# B&R Automation Studio project FASTorySystems (part 3)

### IoMap.iom - 5APC4100_TGL2_000/IoMap.iom
```iecst
VAR_CONFIG
	Cyclic#1.::gCommInput.Array[0] AT %IW."8FLM01.0000.00I-1".EPL_FB_IN_0_I2007_S01;
	Cyclic#1.::gCommInput.Array[1] AT %IW."8FLM01.0000.00I-1".EPL_FB_IN_1_I2007_S02;
	Cyclic#1.::gCommInput.Array[2] AT %IW."8FLM01.0000.00I-1".EPL_FB_IN_2_I2007_S03;
	Cyclic#1.::gCommInput.Array[3] AT %IW."8FLM01.0000.00I-1".EPL_FB_IN_3_I2007_S04;
	Cyclic#1.::gCommInput.Array[4] AT %IW."8FLM01.0000.00I-1".EPL_FB_IN_4_I2007_S05;
	Cyclic#1.::gCommInput.Array[5] AT %IW."8FLM01.0000.00I-1".EPL_FB_IN_5_I2007_S06;
	Cyclic#1.::gCommInput.Array[6] AT %IW."8FLM01.0000.00I-1".EPL_FB_IN_6_I2007_S07;
	Cyclic#1.::gCommInput.Array[7] AT %IW."8FLM01.0000.00I-1".EPL_FB_IN_7_I2007_S08;
	Cyclic#1.::gCommInput.Array[8] AT %IW."8FLM01.0000.00I-1".EPL_FB_IN_8_I2007_S09;
	Cyclic#1.::gCommInput.Array[9] AT %IW."8FLM01.0000.00I-1".EPL_FB_IN_9_I2007_S0A;
	Cyclic#1.::gCommInput.Array[10] AT %IW."8FLM01.0000.00I-1".EPL_FB_IN_10_I2007_S0B;
	Cyclic#1.::gCommInput.Array[11] AT %IW."8FLM01.0000.00I-1".EPL_FB_IN_11_I2007_S0C;
	Cyclic#1.::gCommInput.Array[12] AT %IW."8FLM01.0000.00I-1".EPL_FB_IN_12_I2007_S0D;
	Cyclic#1.::gCommInput.Array[13] AT %IW."8FLM01.0000.00I-1".EPL_FB_IN_13_I2007_S0E;
	Cyclic#1.::gCommInput.Array[14] AT %IW."8FLM01.0000.00I-1".EPL_FB_IN_14_I2007_S0F;
	Cyclic#1.::gCommInput.Array[15] AT %IW."8FLM01.0000.00I-1".EPL_FB_IN_15_I2007_S10;
	Cyclic#1.::gCommInput.Array[16] AT %IW."8FLM01.0000.00I-1".EPL_FB_IN_16_I2007_S11;
	Cyclic#1.::gCommInput.Array[17] AT %IW."8FLM01.0000.00I-1".EPL_FB_IN_17_I2007_S12;
	Cyclic#1.::gCommInput.Array[18] AT %IW."8FLM01.0000.00I-1".EPL_FB_IN_18_I2007_S13;
	Cyclic#1.::gCommInput.Array[19] AT %IW."8FLM01.0000.00I-1".EPL_FB_IN_19_I2007_S14;
	Cyclic#1.::gCommInput.Array[20] AT %IW."8FLM01.0000.00I-1".EPL_FB_IN_20_I2007_S15;
	Cyclic#1.::gCommInput.Array[21] AT %IW."8FLM01.0000.00I-1".EPL_FB_IN_21_I2007_S16;
	Cyclic#1.::gCommInput.Array[22] AT %IW."8FLM01.0000.00I-1".EPL_FB_IN_22_I2007_S17;
	Cyclic#1.::gCommInput.Array[23] AT %IW."8FLM01.0000.00I-1".EPL_FB_IN_23_I2007_S18;
	Cyclic#1.::gCommInput.Array[24] AT %IW."8FLM01.0000.00I-1".EPL_FB_IN_24_I2007_S19;
	Cyclic#1.::gCommInput.Array[25] AT %IW."8FLM01.0000.00I-1".EPL_FB_IN_25_I2007_S1A;
	Cyclic#1.::gCommInput.Array[26] AT %IW."8FLM01.0000.00I-1".EPL_FB_IN_26_I2007_S1B;
	Cyclic#1.::gCommInput.Array[27] AT %IW."8FLM01.0000.00I-1".EPL_FB_IN_27_I2007_S1C;
	Cyclic#1.::gCommInput.Array[28] AT %IW."8FLM01.0000.00I-1".EPL_FB_IN_28_I2007_S1D;
	Cyclic#1.::gCommInput.Array[29] AT %IW."8FLM01.0000.00I-1".EPL_FB_IN_29_I2007_S1E;
	Cyclic#1.::gCommInput.Array[30] AT %IW."8FLM01.0000.00I-1".EPL_FB_IN_30_I2007_S1F;
	Cyclic#1.::gCommInput.Array[31] AT %IW."8FLM01.0000.00I-1".EPL_FB_IN_31_I2007_S20;
	Cyclic#1.::gCommInput.Array[32] AT %IW."8FLM01.0000.00I-1".EPL_FB_IN_32_I2007_S21;
	Cyclic#1.::gCommInput.Array[33] AT %IW."8FLM01.0000.00I-1".EPL_FB_IN_33_I2007_S22;
	Cyclic#1.::gCommInput.Array[34] AT %IW."8FLM01.0000.00I-1".EPL_FB_IN_34_I2007_S23;
	Cyclic#1.::gCommInput.Array[35] AT %IW."8FLM01.0000.00I-1".EPL_FB_IN_35_I2007_S24;
	Cyclic#1.::gCommInput.Array[36] AT %IW."8FLM01.0000.00I-1".EPL_FB_IN_36_I2007_S25;
	Cyclic#1.::gCommInput.Array[37] AT %IW."8FLM01.0000.00I-1".EPL_FB_IN_37_I2007_S26;
	Cyclic#1.::gCommInput.Array[38] AT %IW."8FLM01.0000.00I-1".EPL_FB_IN_38_I2007_S27;
	Cyclic#1.::gCommInput.Array[39] AT %IW."8FLM01.0000.00I-1".EPL_FB_IN_39_I2007_S28;
	Cyclic#1.::gCommInput.Array[40] AT %IW."8FLM01.0000.00I-1".EPL_FB_IN_40_I2007_S29;
	Cyclic#1.::gCommInput.Array[41] AT %IW."8FLM01.0000.00I-1".EPL_FB_IN_41_I2007_S2A;
	Cyclic#1.::gCommInput.Array[42] AT %IW."8FLM01.0000.00I-1".EPL_FB_IN_42_I2007_S2B;
	Cyclic#1.::gCommInput.Array[43] AT %IW."8FLM01.0000.00I-1".EPL_FB_IN_43_I2007_S2C;
	Cyclic#1.::gCommInput.Array[44] AT %IW."8FLM01.0000.00I-1".EPL_FB_IN_44_I2007_S2D;
	Cyclic#1.::gCommInput.Array[45] AT %IW."8FLM01.0000.00I-1".EPL_FB_IN_45_I2007_S2E;
	Cyclic#1.::gCommInput.Array[46] AT %IW."8FLM01.0000.00I-1".EPL_FB_IN_46_I2007_S2F;
	Cyclic#1.::gCommInput.Array[47] AT %IW."8FLM01.0000.00I-1".EPL_FB_IN_47_I2007_S30;
	Cyclic#1.::gCommInput.Array[48] AT %IW."8FLM01.0000.00I-1".EPL_FB_IN_48_I2007_S31;
	Cyclic#1.::gCommInput.Array[49] AT %IW."8FLM01.0000.00I-1".EPL_FB_IN_49_I2007_S32;
	Cyclic#1.::gCommInput.Array[50] AT %IW."8FLM01.0000.00I-1".EPL_FB_IN_50_I2007_S33;
	Cyclic#1.::gCommInput.Array[51] AT %IW."8FLM01.0000.00I-1".EPL_FB_IN_51_I2007_S34;
	Cyclic#1.::gCommInput.Array[52] AT %IW."8FLM01.0000.00I-1".EPL_FB_IN_52_I2007_S35;
	Cyclic#1.::gCommInput.Array[53] AT %IW."8FLM01.0000.00I-1".EPL_FB_IN_53_I2007_S36;
	Cyclic#1.::gCommInput.Array[54] AT %IW."8FLM01.0000.00I-1".EPL_FB_IN_54_I2007_S37;
	Cyclic#1.::gCommInput.Array[55] AT %IW."8FLM01.0000.00I-1".EPL_FB_IN_55_I2007_S38;
	Cyclic#1.::gCommInput.Array[56] AT %IW."8FLM01.0000.00I-1".EPL_FB_IN_56_I2007_S39;
	Cyclic#1.::gCommInput.Array[57] AT %IW."8FLM01.0000.00I-1".EPL_FB_IN_57_I2007_S3A;
	Cyclic#1.::gCommInput.Array[58] AT %IW."8FLM01.0000.00I-1".EPL_FB_IN_58_I2007_S3B;
	Cyclic#1.::gCommInput.Array[59] AT %IW."8FLM01.0000.00I-1".EPL_FB_IN_59_I2007_S3C;
	Cyclic#1.::gCommInput.Array[60] AT %IW."8FLM01.0000.00I-1".EPL_FB_IN_60_I2007_S3D;
	Cyclic#1.::gCommInput.Array[61] AT %IW."8FLM01.0000.00I-1".EPL_FB_IN_61_I2007_S3E;
	Cyclic#1.::gCommInput.Array[62] AT %IW."8FLM01.0000.00I-1".EPL_FB_IN_62_I2007_S3F;
	Cyclic#1.::gCommInput.Array[63] AT %IW."8FLM01.0000.00I-1".EPL_FB_IN_63_I2007_S40;
	Cyclic#1.::gCommInput.Array[64] AT %IW."8FLM01.0000.00I-1".EPL_FB_IN_64_I2007_S41;
	Cyclic#1.::gCommInput.Array[65] AT %IW."8FLM01.0000.00I-1".EPL_FB_IN_65_I2007_S42;
	Cyclic#1.::gCommInput.Array[66] AT %IW."8FLM01.0000.00I-1".EPL_FB_IN_66_I2007_S43;
	Cyclic#1.::gCommInput.Array[67] AT %IW."8FLM01.0000.00I-1".EPL_FB_IN_67_I2007_S44;
	Cyclic#1.::gCommInput.Array[68] AT %IW."8FLM01.0000.00I-1".EPL_FB_IN_68_I2007_S45;
	Cyclic#1.::gCommInput.Array[69] AT %IW."8FLM01.0000.00I-1".EPL_FB_IN_69_I2007_S46;
	Cyclic#1.::gCommInput.Array[70] AT %IW."8FLM01.0000.00I-1".EPL_FB_IN_70_I2007_S47;
	Cyclic#1.::gCommInput.Array[71] AT %IW."8FLM01.0000.00I-1".EPL_FB_IN_71_I2007_S48;
	Cyclic#1.::gCommInput.Array[72] AT %IW."8FLM01.0000.00I-1".EPL_FB_IN_72_I2007_S49;
	Cyclic#1.::gCommInput.Array[73] AT %IW."8FLM01.0000.00I-1".EPL_FB_IN_73_I2007_S4A;
	Cyclic#1.::gCommInput.Array[74] AT %IW."8FLM01.0000.00I-1".EPL_FB_IN_74_I2007_S4B;
	Cyclic#1.::gCommInput.Array[75] AT %IW."8FLM01.0000.00I-1".EPL_FB_IN_75_I2007_S4C;
	Cyclic#1.::gCommInput.Array[76] AT %IW."8FLM01.0000.00I-1".EPL_FB_IN_76_I2007_S4D;
	Cyclic#1.::gCommInput.Array[77] AT %IW."8FLM01.0000.00I-1".EPL_FB_IN_77_I2007_S4E;
	Cyclic#1.::gCommInput.Array[78] AT %IW."8FLM01.0000.00I-1".EPL_FB_IN_78_I2007_S4F;
	Cyclic#1.::gCommInput.Array[79] AT %IW."8FLM01.0000.00I-1".EPL_FB_IN_79_I2007_S50;
	Cyclic#1.::gCommInput.Array[80] AT %IW."8FLM01.0000.00I-1".EPL_FB_IN_80_I2007_S51;
	Cyclic#1.::gCommInput.Array[81] AT %IW."8FLM01.0000.00I-1".EPL_FB_IN_81_I2007_S52;
	Cyclic#1.::gCommInput.Array[82] AT %IW."8FLM01.0000.00I-1".EPL_FB_IN_82_I2007_S53;
	Cyclic#1.::gCommInput.Array[83] AT %IW."8FLM01.0000.00I-1".EPL_FB_IN_83_I2007_S54;
	Cyclic#1.::gCommInput.Array[84] AT %IW."8FLM01.0000.00I-1".EPL_FB_IN_84_I2007_S55;
	Cyclic#1.::gCommInput.Array[85] AT %IW."8FLM01.0000.00I-1".EPL_FB_IN_85_I2007_S56;
	Cyclic#1.::gCommInput.Array[86] AT %IW."8FLM01.0000.00I-1".EPL_FB_IN_86_I2007_S57;
	Cyclic#1.::gCommInput.Array[87] AT %IW."8FLM01.0000.00I-1".EPL_FB_IN_87_I2007_S58;
	Cyclic#1.::gCommInput.Array[88] AT %IW."8FLM01.0000.00I-1".EPL_FB_IN_88_I2007_S59;
	Cyclic#1.::gCommInput.Array[89] AT %IW."8FLM01.0000.00I-1".EPL_FB_IN_89_I2007_S5A;
	Cyclic#1.::gCommInput.Array[90] AT %IW."8FLM01.0000.00I-1".EPL_FB_IN_90_I2007_S5B;
	Cyclic#1.::gCommInput.Array[91] AT %IW."8FLM01.0000.00I-1".EPL_FB_IN_91_I2007_S5C;
	Cyclic#1.::gCommInput.Array[92] AT %IW."8FLM01.0000.00I-1".EPL_FB_IN_92_I2007_S5D;
	Cyclic#1.::gCommInput.Array[93] AT %IW."8FLM01.0000.00I-1".EPL_FB_IN_93_I2007_S5E;
	Cyclic#1.::gCommInput.Array[94] AT %IW."8FLM01.0000.00I-1".EPL_FB_IN_94_I2007_S5F;
	Cyclic#1.::gCommInput.Array[95] AT %IW."8FLM01.0000.00I-1".EPL_FB_IN_95_I2007_S60;
	Cyclic#1.::gCommInput.Array[96] AT %IW."8FLM01.0000.00I-1".EPL_FB_IN_96_I2007_S61;
	Cyclic#1.::gCommInput.Array[97] AT %IW."8FLM01.0000.00I-1".EPL_FB_IN_97_I2007_S62;
	Cyclic#1.::gCommInput.Array[98] AT %IW."8FLM01.0000.00I-1".EPL_FB_IN_98_I2007_S63;
	Cyclic#1.::gCommInput.Array[99] AT %IW."8FLM01.0000.00I-1".EPL_FB_IN_99_I2007_S64;
	Cyclic#1.::gCommInput.Array[100] AT %IW."8FLM01.0000.00I-1".EPL_FB_IN_100_I2007_S65;
	Cyclic#1.::gCommInput.Array[101] AT %IW."8FLM01.0000.00I-1".EPL_FB_IN_101_I2007_S66;
	Cyclic#1.::gCommInput.Array[102] AT %IW."8FLM01.0000.00I-1".EPL_FB_IN_102_I2007_S67;
	Cyclic#1.::gCommInput.Array[103] AT %IW."8FLM01.0000.00I-1".EPL_FB_IN_103_I2007_S68;
	Cyclic#1.::gCommInput.Array[104] AT %IW."8FLM01.0000.00I-1".EPL_FB_IN_104_I2007_S69;
	Cyclic#1.::gCommInput.Array[105] AT %IW."8FLM01.0000.00I-1".EPL_FB_IN_105_I2007_S6A;
	Cyclic#1.::gCommInput.Array[106] AT %IW."8FLM01.0000.00I-1".EPL_FB_IN_106_I2007_S6B;
	Cyclic#1.::gCommInput.Array[107] AT %IW."8FLM01.0000.00I-1".EPL_FB_IN_107_I2007_S6C;
	Cyclic#1.::gCommInput.Array[108] AT %IW."8FLM01.0000.00I-1".EPL_FB_IN_108_I2007_S6D;
	Cyclic#1.::gCommInput.Array[109] AT %IW."8FLM01.0000.00I-1".EPL_FB_IN_109_I2007_S6E;
	Cyclic#1.::gCommInput.Array[110] AT %IW."8FLM01.0000.00I-1".EPL_FB_IN_110_I2007_S6F;
	Cyclic#1.::gCommInput.Array[111] AT %IW."8FLM01.0000.00I-1".EPL_FB_IN_111_I2007_S70;
	Cyclic#1.::gCommInput.Array[112] AT %IW."8FLM01.0000.00I-1".EPL_FB_IN_112_I2007_S71;
	Cyclic#1.::gCommInput.Array[113] AT %IW."8FLM01.0000.00I-1".EPL_FB_IN_113_I2007_S72;
	Cyclic#1.::gCommInput.Array[114] AT %IW."8FLM01.0000.00I-1".EPL_FB_IN_114_I2007_S73;
	Cyclic#1.::gCommInput.Array[115] AT %IW."8FLM01.0000.00I-1".EPL_FB_IN_115_I2007_S74;
	Cyclic#1.::gCommInput.Array[116] AT %IW."8FLM01.0000.00I-1".EPL_FB_IN_116_I2007_S75;
	Cyclic#1.::gCommInput.Array[117] AT %IW."8FLM01.0000.00I-1".EPL_FB_IN_117_I2007_S76;
	Cyclic#1.::gCommInput.Array[118] AT %IW."8FLM01.0000.00I-1".EPL_FB_IN_118_I2007_S77;
	Cyclic#1.::gCommInput.Array[119] AT %IW."8FLM01.0000.00I-1".EPL_FB_IN_119_I2007_S78;
	Cyclic#1.::gCommInput.Array[120] AT %IW."8FLM01.0000.00I-1".EPL_FB_IN_120_I2007_S79;
	Cyclic#1.::gCommInput.Array[121] AT %IW."8FLM01.0000.00I-1".EPL_FB_IN_121_I2007_S7A;
	Cyclic#1.::gCommInput.Array[122] AT %IW."8FLM01.0000.00I-1".EPL_FB_IN_122_I2007_S7B;
	Cyclic#1.::gCommInput.Array[123] AT %IW."8FLM01.0000.00I-1".EPL_FB_IN_123_I2007_S7C;
	Cyclic#1.::gCommInput.Array[124] AT %IW."8FLM01.0000.00I-1".EPL_FB_IN_124_I2007_S7D;
	Cyclic#1.::gCommInput.Array[125] AT %IW."8FLM01.0000.00I-1".EPL_FB_IN_125_I2007_S7E;
	Cyclic#1.::gCommInput.Array[126] AT %IW."8FLM01.0000.00I-1".EPL_FB_IN_126_I2007_S7F;
	Cyclic#1.::gCommInput.Array[127] AT %IW."8FLM01.0000.00I-1".EPL_FB_IN_127_I2007_S80;
	Cyclic#1.::gCommInput.Array[128] AT %IW."8FLM01.0000.00I-1".EPL_FB_IN_128_I2007_S81;
	Cyclic#1.::gCommInput.Array[129] AT %IW."8FLM01.0000.00I-1".EPL_FB_IN_129_I2007_S82;
	Cyclic#1.::gCommInput.Array[130] AT %IW."8FLM01.0000.00I-1".EPL_FB_IN_130_I2007_S83;
	Cyclic#1.::gCommInput.Array[131] AT %IW."8FLM01.0000.00I-1".EPL_FB_IN_131_I2007_S84;
	Cyclic#1.::gCommInput.Array[132] AT %IW."8FLM01.0000.00I-1".EPL_FB_IN_132_I2007_S85;
	Cyclic#1.::gCommInput.Array[133] AT %IW."8FLM01.0000.00I-1".EPL_FB_IN_133_I2007_S86;
	Cyclic#1.::gCommInput.Array[134] AT %IW."8FLM01.0000.00I-1".EPL_FB_IN_134_I2007_S87;
	Cyclic#1.::gCommInput.Array[135] AT %IW."8FLM01.0000.00I-1".EPL_FB_IN_135_I2007_S88;
	Cyclic#1.::gCommInput.Array[136] AT %IW."8FLM01.0000.00I-1".EPL_FB_IN_136_I2007_S89;
	Cyclic#1.::gCommInput.Array[137] AT %IW."8FLM01.0000.00I-1".EPL_FB_IN_137_I2007_S8A;
	Cyclic#1.::gCommInput.Array[138] AT %IW."8FLM01.0000.00I-1".EPL_FB_IN_138_I2007_S8B;
	Cyclic#1.::gCommInput.Array[139] AT %IW."8FLM01.0000.00I-1".EPL_FB_IN_139_I2007_S8C;
	Cyclic#1.::gCommInput.Array[140] AT %IW."8FLM01.0000.00I-1".EPL_FB_IN_140_I2007_S8D;
	Cyclic#1.::gCommInput.Array[141] AT %IW."8FLM01.0000.00I-1".EPL_FB_IN_141_I2007_S8E;
	Cyclic#1.::gCommInput.Array[142] AT %IW."8FLM01.0000.00I-1".EPL_FB_IN_142_I2007_S8F;
	Cyclic#1.::gCommInput.Array[143] AT %IW."8FLM01.0000.00I-1".EPL_FB_IN_143_I2007_S90;
	Cyclic#1.::gCommInput.Array[144] AT %IW."8FLM01.0000.00I-1".EPL_FB_IN_144_I2007_S91;
	Cyclic#1.::gCommInput.Array[145] AT %IW."8FLM01.0000.00I-1".EPL_FB_IN_145_I2007_S92;
	Cyclic#1.::gCommInput.Array[146] AT %IW."8FLM01.0000.00I-1".EPL_FB_IN_146_I2007_S93;
	Cyclic#1.::gCommInput.Array[147] AT %IW."8FLM01.0000.00I-1".EPL_FB_IN_147_I2007_S94;
	Cyclic#1.::gCommInput.Array[148] AT %IW."8FLM01.0000.00I-1".EPL_FB_IN_148_I2007_S95;
	Cyclic#1.::gCommInput.Array[149] AT %IW."8FLM01.0000.00I-1".EPL_FB_IN_149_I2007_S96;
	Cyclic#1.::gCommInput.Array[150] AT %IW."8FLM01.0000.00I-1".EPL_FB_IN_150_I2007_S97;
	Cyclic#1.::gCommInput.Array[151] AT %IW."8FLM01.0000.00I-1".EPL_FB_IN_151_I2007_S98;
	Cyclic#1.::gCommInput.Array[152] AT %IW."8FLM01.0000.00I-1".EPL_FB_IN_152_I2007_S99;
	Cyclic#1.::gCommInput.Array[153] AT %IW."8FLM01.0000.00I-1".EPL_FB_IN_153_I2007_S9A;
	Cyclic#1.::gCommInput.Array[154] AT %IW."8FLM01.0000.00I-1".EPL_FB_IN_154_I2007_S9B;
	Cyclic#1.::gCommInput.Array[155] AT %IW."8FLM01.0000.00I-1".EPL_FB_IN_155_I2007_S9C;
	Cyclic#1.::gCommInput.Array[156] AT %IW."8FLM01.0000.00I-1".EPL_FB_IN_156_I2007_S9D;
	Cyclic#1.::gCommInput.Array[157] AT %IW."8FLM01.0000.00I-1".EPL_FB_IN_157_I2007_S9E;
	Cyclic#1.::gCommInput.Array[158] AT %IW."8FLM01.0000.00I-1".EPL_FB_IN_158_I2007_S9F;
	Cyclic#1.::gCommInput.Array[159] AT %IW."8FLM01.0000.00I-1".EPL_FB_IN_159_I2007_SA0;
	Cyclic#1.::gCommInput.Array[160] AT %IW."8FLM01.0000.00I-1".EPL_FB_IN_160_I2007_SA1;
	Cyclic#1.::gCommInput.Array[161] AT %IW."8FLM01.0000.00I-1".EPL_FB_IN_161_I2007_SA2;
	Cyclic#1.::gCommInput.Array[162] AT %IW."8FLM01.0000.00I-1".EPL_FB_IN_162_I2007_SA3;
	Cyclic#1.::gCommInput.Array[163] AT %IW."8FLM01.0000.00I-1".EPL_FB_IN_163_I2007_SA4;
	Cyclic#1.::gCommInput.Array[164] AT %IW."8FLM01.0000.00I-1".EPL_FB_IN_164_I2007_SA5;
	Cyclic#1.::gCommInput.Array[165] AT %IW."8FLM01.0000.00I-1".EPL_FB_IN_165_I2007_SA6;
	Cyclic#1.::gCommInput.Array[166] AT %IW."8FLM01.0000.00I-1".EPL_FB_IN_166_I2007_SA7;
	Cyclic#1.::gCommInput.Array[167] AT %IW."8FLM01.0000.00I-1".EPL_FB_IN_167_I2007_SA8;
	Cyclic#1.::gCommInput.Array[168] AT %IW."8FLM01.0000.00I-1".EPL_FB_IN_168_I2007_SA9;
	Cyclic#1.::gCommInput.Array[169] AT %IW."8FLM01.0000.00I-1".EPL_FB_IN_169_I2007_SAA;
	Cyclic#1.::gCommInput.Array[170] AT %IW."8FLM01.0000.00I-1".EPL_FB_IN_170_I2007_SAB;
	Cyclic#1.::gCommInput.Array[171] AT %IW."8FLM01.0000.00I-1".EPL_FB_IN_171_I2007_SAC;
	Cyclic#1.::gCommInput.Array[172] AT %IW."8FLM01.0000.00I-1".EPL_FB_IN_172_I2007_SAD;
	Cyclic#1.::gCommInput.Array[173] AT %IW."8FLM01.0000.00I-1".EPL_FB_IN_173_I2007_SAE;
	Cyclic#1.::gCommInput.Array[174] AT %IW."8FLM01.0000.00I-1".EPL_FB_IN_174_I2007_SAF;
	Cyclic#1.::gCommInput.Array[175] AT %IW."8FLM01.0000.00I-1".EPL_FB_IN_175_I2007_SB0;
	Cyclic#1.::gCommInput.Array[176] AT %IW."8FLM01.0000.00I-1".EPL_FB_IN_176_I2007_SB1;
	Cyclic#1.::gCommInput.Array[177] AT %IW."8FLM01.0000.00I-1".EPL_FB_IN_177_I2007_SB2;
	Cyclic#1.::gCommInput.Array[178] AT %IW."8FLM01.0000.00I-1".EPL_FB_IN_178_I2007_SB3;
	Cyclic#1.::gCommInput.Array[179] AT %IW."8FLM01.0000.00I-1".EPL_FB_IN_179_I2007_SB4;
	Cyclic#1.::gCommInput.Array[180] AT %IW."8FLM01.0000.00I-1".EPL_FB_IN_180_I2007_SB5;
	Cyclic#1.::gCommInput.Array[181] AT %IW."8FLM01.0000.00I-1".EPL_FB_IN_181_I2007_SB6;
	Cyclic#1.::gCommInput.Array[182] AT %IW."8FLM01.0000.00I-1".EPL_FB_IN_182_I2007_SB7;
	Cyclic#1.::gCommInput.Array[183] AT %IW."8FLM01.0000.00I-1".EPL_FB_IN_183_I2007_SB8;
	Cyclic#1.::gCommInput.Array[184] AT %IW."8FLM01.0000.00I-1".EPL_FB_IN_184_I2007_SB9;
	Cyclic#1.::gCommInput.Array[185] AT %IW."8FLM01.0000.00I-1".EPL_FB_IN_185_I2007_SBA;
	Cyclic#1.::gCommInput.Array[186] AT %IW."8FLM01.0000.00I-1".EPL_FB_IN_186_I2007_SBB;
	Cyclic#1.::gCommInput.Array[187] AT %IW."8FLM01.0000.00I-1".EPL_FB_IN_187_I2007_SBC;
	Cyclic#1.::gCommInput.Array[188] AT %IW."8FLM01.0000.00I-1".EPL_FB_IN_188_I2007_SBD;
	Cyclic#1.::gCommInput.Array[189] AT %IW."8FLM01.0000.00I-1".EPL_FB_IN_189_I2007_SBE;
	Cyclic#1.::gCommInput.Array[190] AT %IW."8FLM01.0000.00I-1".EPL_FB_IN_190_I2007_SBF;
	Cyclic#1.::gCommInput.Array[191] AT %IW."8FLM01.0000.00I-1".EPL_FB_IN_191_I2007_SC0;
	Cyclic#1.::gCommInput.Array[192] AT %IW."8FLM01.0000.00I-1".EPL_FB_IN_192_I2007_SC1;
	Cyclic#1.::gCommInput.Array[193] AT %IW."8FLM01.0000.00I-1".EPL_FB_IN_193_I2007_SC2;
	Cyclic#1.::gCommInput.Array[194] AT %IW."8FLM01.0000.00I-1".EPL_FB_IN_194_I2007_SC3;
	Cyclic#1.::gCommInput.Array[195] AT %IW."8FLM01.0000.00I-1".EPL_FB_IN_195_I2007_SC4;
	Cyclic#1.::gCommInput.Array[196] AT %IW."8FLM01.0000.00I-1".EPL_FB_IN_196_I2007_SC5;
	Cyclic#1.::gCommInput.Array[197] AT %IW."8FLM01.0000.00I-1".EPL_FB_IN_197_I2007_SC6;
	Cyclic#1.::gCommInput.Array[198] AT %IW."8FLM01.0000.00I-1".EPL_FB_IN_198_I2007_SC7;
	Cyclic#1.::gCommInput.Array[199] AT %IW."8FLM01.0000.00I-1".EPL_FB_IN_199_I2007_SC8;
	Cyclic#1.::gCommOutput.Array[0] AT %QW."8FLM01.0000.00I-1".EPL_FB_OUT_0_I2008_S01Out;
	Cyclic#1.::gCommOutput.Array[1] AT %QW."8FLM01.0000.00I-1".EPL_FB_OUT_1_I2008_S02Out;
	Cyclic#1.::gCommOutput.Array[2] AT %QW."8FLM01.0000.00I-1".EPL_FB_OUT_2_I2008_S03Out;
	Cyclic#1.::gCommOutput.Array[3] AT %QW."8FLM01.0000.00I-1".EPL_FB_OUT_3_I2008_S04Out;
	Cyclic#1.::gCommOutput.Array[4] AT %QW."8FLM01.0000.00I-1".EPL_FB_OUT_4_I2008_S05Out;
	Cyclic#1.::gCommOutput.Array[5] AT %QW."8FLM01.0000.00I-1".EPL_FB_OUT_5_I2008_S06Out;
	Cyclic#1.::gCommOutput.Array[6] AT %QW."8FLM01.0000.00I-1".EPL_FB_OUT_6_I2008_S07Out;
	Cyclic#1.::gCommOutput.Array[7] AT %QW."8FLM01.0000.00I-1".EPL_FB_OUT_7_I2008_S08Out;
	Cyclic#1.::gCommOutput.Array[8] AT %QW."8FLM01.0000.00I-1".EPL_FB_OUT_8_I2008_S09Out;
	Cyclic#1.::gCommOutput.Array[9] AT %QW."8FLM01.0000.00I-1".EPL_FB_OUT_9_I2008_S0AOut;
	Cyclic#1.::gCommOutput.Array[10] AT %QW."8FLM01.0000.00I-1".EPL_FB_OUT_10_I2008_S0BOut;
	Cyclic#1.::gCommOutput.Array[11] AT %QW."8FLM01.0000.00I-1".EPL_FB_OUT_11_I2008_S0COut;
	Cyclic#1.::gCommOutput.Array[12] AT %QW."8FLM01.0000.00I-1".EPL_FB_OUT_12_I2008_S0DOut;
	Cyclic#1.::gCommOutput.Array[13] AT %QW."8FLM01.0000.00I-1".EPL_FB_OUT_13_I2008_S0EOut;
	Cyclic#1.::gCommOutput.Array[14] AT %QW."8FLM01.0000.00I-1".EPL_FB_OUT_14_I2008_S0FOut;
	Cyclic#1.::gCommOutput.Array[15] AT %QW."8FLM01.0000.00I-1".EPL_FB_OUT_15_I2008_S10Out;
	Cyclic#1.::gCommOutput.Array[16] AT %QW."8FLM01.0000.00I-1".EPL_FB_OUT_16_I2008_S11Out;
	Cyclic#1.::gCommOutput.Array[17] AT %QW."8FLM01.0000.00I-1".EPL_FB_OUT_17_I2008_S12Out;
	Cyclic#1.::gCommOutput.Array[18] AT %QW."8FLM01.0000.00I-1".EPL_FB_OUT_18_I2008_S13Out;
	Cyclic#1.::gCommOutput.Array[19] AT %QW."8FLM01.0000.00I-1".EPL_FB_OUT_19_I2008_S14Out;
	Cyclic#1.::gCommOutput.Array[20] AT %QW."8FLM01.0000.00I-1".EPL_FB_OUT_20_I2008_S15Out;
	Cyclic#1.::gCommOutput.Array[21] AT %QW."8FLM01.0000.00I-1".EPL_FB_OUT_21_I2008_S16Out;
	Cyclic#1.::gCommOutput.Array[22] AT %QW."8FLM01.0000.00I-1".EPL_FB_OUT_22_I2008_S17Out;
	Cyclic#1.::gCommOutput.Array[23] AT %QW."8FLM01.0000.00I-1".EPL_FB_OUT_23_I2008_S18Out;
	Cyclic#1.::gCommOutput.Array[24] AT %QW."8FLM01.0000.00I-1".EPL_FB_OUT_24_I2008_S19Out;
	Cyclic#1.::gCommOutput.Array[25] AT %QW."8FLM01.0000.00I-1".EPL_FB_OUT_25_I2008_S1AOut;
	Cyclic#1.::gCommOutput.Array[26] AT %QW."8FLM01.0000.00I-1".EPL_FB_OUT_26_I2008_S1BOut;
	Cyclic#1.::gCommOutput.Array[27] AT %QW."8FLM01.0000.00I-1".EPL_FB_OUT_27_I2008_S1COut;
	Cyclic#1.::gCommOutput.Array[28] AT %QW."8FLM01.0000.00I-1".EPL_FB_OUT_28_I2008_S1DOut;
	Cyclic#1.::gCommOutput.Array[29] AT %QW."8FLM01.0000.00I-1".EPL_FB_OUT_29_I2008_S1EOut;
	Cyclic#1.::gCommOutput.Array[30] AT %QW."8FLM01.0000.00I-1".EPL_FB_OUT_30_I2008_S1FOut;
	Cyclic#1.::gCommOutput.Array[31] AT %QW."8FLM01.0000.00I-1".EPL_FB_OUT_31_I2008_S20Out;
	Cyclic#1.::gCommOutput.Array[32] AT %QW."8FLM01.0000.00I-1".EPL_FB_OUT_32_I2008_S21Out;
	Cyclic#1.::gCommOutput.Array[33] AT %QW."8FLM01.0000.00I-1".EPL_FB_OUT_33_I2008_S22Out;
	Cyclic#1.::gCommOutput.Array[34] AT %QW."8FLM01.0000.00I-1".EPL_FB_OUT_34_I2008_S23Out;
	Cyclic#1.::gCommOutput.Array[35] AT %QW."8FLM01.0000.00I-1".EPL_FB_OUT_35_I2008_S24Out;
	Cyclic#1.::gCommOutput.Array[36] AT %QW."8FLM01.0000.00I-1".EPL_FB_OUT_36_I2008_S25Out;
	Cyclic#1.::gCommOutput.Array[37] AT %QW."8FLM01.0000.00I-1".EPL_FB_OUT_37_I2008_S26Out;
	Cyclic#1.::gCommOutput.Array[38] AT %QW."8FLM01.0000.00I-1".EPL_FB_OUT_38_I2008_S27Out;
	Cyclic#1.::gCommOutput.Array[39] AT %QW."8FLM01.0000.00I-1".EPL_FB_OUT_39_I2008_S28Out;
	Cyclic#1.::gCommOutput.Array[40] AT %QW."8FLM01.0000.00I-1".EPL_FB_OUT_40_I2008_S29Out;
	Cyclic#1.::gCommOutput.Array[41] AT %QW."8FLM01.0000.00I-1".EPL_FB_OUT_41_I2008_S2AOut;
	Cyclic#1.::gCommOutput.Array[42] AT %QW."8FLM01.0000.00I-1".EPL_FB_OUT_42_I2008_S2BOut;
	Cyclic#1.::gCommOutput.Array[43] AT %QW."8FLM01.0000.00I-1".EPL_FB_OUT_43_I2008_S2COut;
	Cyclic#1.::gCommOutput.Array[44] AT %QW."8FLM01.0000.00I-1".EPL_FB_OUT_44_I2008_S2DOut;
	Cyclic#1.::gCommOutput.Array[45] AT %QW."8FLM01.0000.00I-1".EPL_FB_OUT_45_I2008_S2EOut;
	Cyclic#1.::gCommOutput.Array[46] AT %QW."8FLM01.0000.00I-1".EPL_FB_OUT_46_I2008_S2FOut;
	Cyclic#1.::gCommOutput.Array[47] AT %QW."8FLM01.0000.00I-1".EPL_FB_OUT_47_I2008_S30Out;
	Cyclic#1.::gCommOutput.Array[48] AT %QW."8FLM01.0000.00I-1".EPL_FB_OUT_48_I2008_S31Out;
	Cyclic#1.::gCommOutput.Array[49] AT %QW."8FLM01.0000.00I-1".EPL_FB_OUT_49_I2008_S32Out;
	Cyclic#1.::gCommOutput.Array[50] AT %QW."8FLM01.0000.00I-1".EPL_FB_OUT_50_I2008_S33Out;
	Cyclic#1.::gCommOutput.Array[51] AT %QW."8FLM01.0000.00I-1".EPL_FB_OUT_51_I2008_S34Out;
	Cyclic#1.::gCommOutput.Array[52] AT %QW."8FLM01.0000.00I-1".EPL_FB_OUT_52_I2008_S35Out;
	Cyclic#1.::gCommOutput.Array[53] AT %QW."8FLM01.0000.00I-1".EPL_FB_OUT_53_I2008_S36Out;
	Cyclic#1.::gCommOutput.Array[54] AT %QW."8FLM01.0000.00I-1".EPL_FB_OUT_54_I2008_S37Out;
	Cyclic#1.::gCommOutput.Array[55] AT %QW."8FLM01.0000.00I-1".EPL_FB_OUT_55_I2008_S38Out;
	Cyclic#1.::gCommOutput.Array[56] AT %QW."8FLM01.0000.00I-1".EPL_FB_OUT_56_I2008_S39Out;
	Cyclic#1.::gCommOutput.Array[57] AT %QW."8FLM01.0000.00I-1".EPL_FB_OUT_57_I2008_S3AOut;
	Cyclic#1.::gCommOutput.Array[58] AT %QW."8FLM01.0000.00I-1".EPL_FB_OUT_58_I2008_S3BOut;
	Cyclic#1.::gCommOutput.Array[59] AT %QW."8FLM01.0000.00I-1".EPL_FB_OUT_59_I2008_S3COut;
	Cyclic#1.::gCommOutput.Array[60] AT %QW."8FLM01.0000.00I-1".EPL_FB_OUT_60_I2008_S3DOut;
	Cyclic#1.::gCommOutput.Array[61] AT %QW."8FLM01.0000.00I-1".EPL_FB_OUT_61_I2008_S3EOut;
	Cyclic#1.::gCommOutput.Array[62] AT %QW."8FLM01.0000.00I-1".EPL_FB_OUT_62_I2008_S3FOut;
	Cyclic#1.::gCommOutput.Array[63] AT %QW."8FLM01.0000.00I-1".EPL_FB_OUT_63_I2008_S40Out;
	Cyclic#1.::gCommOutput.Array[64] AT %QW."8FLM01.0000.00I-1".EPL_FB_OUT_64_I2008_S41Out;
	Cyclic#1.::gCommOutput.Array[65] AT %QW."8FLM01.0000.00I-1".EPL_FB_OUT_65_I2008_S42Out;
	Cyclic#1.::gCommOutput.Array[66] AT %QW."8FLM01.0000.00I-1".EPL_FB_OUT_66_I2008_S43Out;
	Cyclic#1.::gCommOutput.Array[67] AT %QW."8FLM01.0000.00I-1".EPL_FB_OUT_67_I2008_S44Out;
	Cyclic#1.::gCommOutput.Array[68] AT %QW."8FLM01.0000.00I-1".EPL_FB_OUT_68_I2008_S45Out;
	Cyclic#1.::gCommOutput.Array[69] AT %QW."8FLM01.0000.00I-1".EPL_FB_OUT_69_I2008_S46Out;
	Cyclic#1.::gCommOutput.Array[70] AT %QW."8FLM01.0000.00I-1".EPL_FB_OUT_70_I2008_S47Out;
	Cyclic#1.::gCommOutput.Array[71] AT %QW."8FLM01.0000.00I-1".EPL_FB_OUT_71_I2008_S48Out;
	Cyclic#1.::gCommOutput.Array[72] AT %QW."8FLM01.0000.00I-1".EPL_FB_OUT_72_I2008_S49Out;
	Cyclic#1.::gCommOutput.Array[73] AT %QW."8FLM01.0000.00I-1".EPL_FB_OUT_73_I2008_S4AOut;
	Cyclic#1.::gCommOutput.Array[74] AT %QW."8FLM01.0000.00I-1".EPL_FB_OUT_74_I2008_S4BOut;
	Cyclic#1.::gCommOutput.Array[75] AT %QW."8FLM01.0000.00I-1".EPL_FB_OUT_75_I2008_S4COut;
	Cyclic#1.::gCommOutput.Array[76] AT %QW."8FLM01.0000.00I-1".EPL_FB_OUT_76_I2008_S4DOut;
	Cyclic#1.::gCommOutput.Array[77] AT %QW."8FLM01.0000.00I-1".EPL_FB_OUT_77_I2008_S4EOut;
	Cyclic#1.::gCommOutput.Array[78] AT %QW."8FLM01.0000.00I-1".EPL_FB_OUT_78_I2008_S4FOut;
	Cyclic#1.::gCommOutput.Array[79] AT %QW."8FLM01.0000.00I-1".EPL_FB_OUT_79_I2008_S50Out;
	Cyclic#1.::gCommOutput.Array[80] AT %QW."8FLM01.0000.00I-1".EPL_FB_OUT_80_I2008_S51Out;
	Cyclic#1.::gCommOutput.Array[81] AT %QW."8FLM01.0000.00I-1".EPL_FB_OUT_81_I2008_S52Out;
	Cyclic#1.::gCommOutput.Array[82] AT %QW."8FLM01.0000.00I-1".EPL_FB_OUT_82_I2008_S53Out;
	Cyclic#1.::gCommOutput.Array[83] AT %QW."8FLM01.0000.00I-1".EPL_FB_OUT_83_I2008_S54Out;
	Cyclic#1.::gCommOutput.Array[84] AT %QW."8FLM01.0000.00I-1".EPL_FB_OUT_84_I2008_S55Out;
	Cyclic#1.::gCommOutput.Array[85] AT %QW."8FLM01.0000.00I-1".EPL_FB_OUT_85_I2008_S56Out;
	Cyclic#1.::gCommOutput.Array[86] AT %QW."8FLM01.0000.00I-1".EPL_FB_OUT_86_I2008_S57Out;
	Cyclic#1.::gCommOutput.Array[87] AT %QW."8FLM01.0000.00I-1".EPL_FB_OUT_87_I2008_S58Out;
	Cyclic#1.::gCommOutput.Array[88] AT %QW."8FLM01.0000.00I-1".EPL_FB_OUT_88_I2008_S59Out;
	Cyclic#1.::gCommOutput.Array[89] AT %QW."8FLM01.0000.00I-1".EPL_FB_OUT_89_I2008_S5AOut;
	Cyclic#1.::gCommOutput.Array[90] AT %QW."8FLM01.0000.00I-1".EPL_FB_OUT_90_I2008_S5BOut;
	Cyclic#1.::gCommOutput.Array[91] AT %QW."8FLM01.0000.00I-1".EPL_FB_OUT_91_I2008_S5COut;
	Cyclic#1.::gCommOutput.Array[92] AT %QW."8FLM01.0000.00I-1".EPL_FB_OUT_92_I2008_S5DOut;
	Cyclic#1.::gCommOutput.Array[93] AT %QW."8FLM01.0000.00I-1".EPL_FB_OUT_93_I2008_S5EOut;
	Cyclic#1.::gCommOutput.Array[94] AT %QW."8FLM01.0000.00I-1".EPL_FB_OUT_94_I2008_S5FOut;
	Cyclic#1.::gCommOutput.Array[95] AT %QW."8FLM01.0000.00I-1".EPL_FB_OUT_95_I2008_S60Out;
	Cyclic#1.::gCommOutput.Array[96] AT %QW."8FLM01.0000.00I-1".EPL_FB_OUT_96_I2008_S61Out;
	Cyclic#1.::gCommOutput.Array[97] AT %QW."8FLM01.0000.00I-1".EPL_FB_OUT_97_I2008_S62Out;
	Cyclic#1.::gCommOutput.Array[98] AT %QW."8FLM01.0000.00I-1".EPL_FB_OUT_98_I2008_S63Out;
	Cyclic#1.::gCommOutput.Array[99] AT %QW."8FLM01.0000.00I-1".EPL_FB_OUT_99_I2008_S64Out;
	Cyclic#1.::gCommOutput.Array[100] AT %QW."8FLM01.0000.00I-1".EPL_FB_OUT_100_I2008_S65Out;
	Cyclic#1.::gCommOutput.Array[101] AT %QW."8FLM01.0000.00I-1".EPL_FB_OUT_101_I2008_S66Out;
	Cyclic#1.::gCommOutput.Array[102] AT %QW."8FLM01.0000.00I-1".EPL_FB_OUT_102_I2008_S67Out;
	Cyclic#1.::gCommOutput.Array[103] AT %QW."8FLM01.0000.00I-1".EPL_FB_OUT_103_I2008_S68Out;
	Cyclic#1.::gCommOutput.Array[104] AT %QW."8FLM01.0000.00I-1".EPL_FB_OUT_104_I2008_S69Out;
	Cyclic#1.::gCommOutput.Array[105] AT %QW."8FLM01.0000.00I-1".EPL_FB_OUT_105_I2008_S6AOut;
	Cyclic#1.::gCommOutput.Array[106] AT %QW."8FLM01.0000.00I-1".EPL_FB_OUT_106_I2008_S6BOut;
	Cyclic#1.::gCommOutput.Array[107] AT %QW."8FLM01.0000.00I-1".EPL_FB_OUT_107_I2008_S6COut;
	Cyclic#1.::gCommOutput.Array[108] AT %QW."8FLM01.0000.00I-1".EPL_FB_OUT_108_I2008_S6DOut;
	Cyclic#1.::gCommOutput.Array[109] AT %QW."8FLM01.0000.00I-1".EPL_FB_OUT_109_I2008_S6EOut;
	Cyclic#1.::gCommOutput.Array[110] AT %QW."8FLM01.0000.00I-1".EPL_FB_OUT_110_I2008_S6FOut;
	Cyclic#1.::gCommOutput.Array[111] AT %QW."8FLM01.0000.00I-1".EPL_FB_OUT_111_I2008_S70Out;
	Cyclic#1.::gCommOutput.Array[112] AT %QW."8FLM01.0000.00I-1".EPL_FB_OUT_112_I2008_S71Out;
	Cyclic#1.::gCommOutput.Array[113] AT %QW."8FLM01.0000.00I-1".EPL_FB_OUT_113_I2008_S72Out;
	Cyclic#1.::gCommOutput.Array[114] AT %QW."8FLM01.0000.00I-1".EPL_FB_OUT_114_I2008_S73Out;
	Cyclic#1.::gCommOutput.Array[115] AT %QW."8FLM01.0000.00I-1".EPL_FB_OUT_115_I2008_S74Out;
	Cyclic#1.::gCommOutput.Array[116] AT %QW."8FLM01.0000.00I-1".EPL_FB_OUT_116_I2008_S75Out;
	Cyclic#1.::gCommOutput.Array[117] AT %QW."8FLM01.0000.00I-1".EPL_FB_OUT_117_I2008_S76Out;
	Cyclic#1.::gCommOutput.Array[118] AT %QW."8FLM01.0000.00I-1".EPL_FB_OUT_118_I2008_S77Out;
	Cyclic#1.::gCommOutput.Array[119] AT %QW."8FLM01.0000.00I-1".EPL_FB_OUT_119_I2008_S78Out;
	Cyclic#1.::gCommOutput.Array[120] AT %QW."8FLM01.0000.00I-1".EPL_FB_OUT_120_I2008_S79Out;
	Cyclic#1.::gCommOutput.Array[121] AT %QW."8FLM01.0000.00I-1".EPL_FB_OUT_121_I2008_S7AOut;
	Cyclic#1.::gCommOutput.Array[122] AT %QW."8FLM01.0000.00I-1".EPL_FB_OUT_122_I2008_S7BOut;
	Cyclic#1.::gCommOutput.Array[123] AT %QW."8FLM01.0000.00I-1".EPL_FB_OUT_123_I2008_S7COut;
	Cyclic#1.::gCommOutput.Array[124] AT %QW."8FLM01.0000.00I-1".EPL_FB_OUT_124_I2008_S7DOut;
	Cyclic#1.::gCommOutput.Array[125] AT %QW."8FLM01.0000.00I-1".EPL_FB_OUT_125_I2008_S7EOut;
	Cyclic#1.::gCommOutput.Array[126] AT %QW."8FLM01.0000.00I-1".EPL_FB_OUT_126_I2008_S7FOut;
	Cyclic#1.::gCommOutput.Array[127] AT %QW."8FLM01.0000.00I-1".EPL_FB_OUT_127_I2008_S80Out;
	Cyclic#1.::gCommOutput.Array[128] AT %QW."8FLM01.0000.00I-1".EPL_FB_OUT_128_I2008_S81Out;
	Cyclic#1.::gCommOutput.Array[129] AT %QW."8FLM01.0000.00I-1".EPL_FB_OUT_129_I2008_S82Out;
	Cyclic#1.::gCommOutput.Array[130] AT %QW."8FLM01.0000.00I-1".EPL_FB_OUT_130_I2008_S83Out;
	Cyclic#1.::gCommOutput.Array[131] AT %QW."8FLM01.0000.00I-1".EPL_FB_OUT_131_I2008_S84Out;
	Cyclic#1.::gCommOutput.Array[132] AT %QW."8FLM01.0000.00I-1".EPL_FB_OUT_132_I2008_S85Out;
	Cyclic#1.::gCommOutput.Array[133] AT %QW."8FLM01.0000.00I-1".EPL_FB_OUT_133_I2008_S86Out;
	Cyclic#1.::gCommOutput.Array[134] AT %QW."8FLM01.0000.00I-1".EPL_FB_OUT_134_I2008_S87Out;
	Cyclic#1.::gCommOutput.Array[135] AT %QW."8FLM01.0000.00I-1".EPL_FB_OUT_135_I2008_S88Out;
	Cyclic#1.::gCommOutput.Array[136] AT %QW."8FLM01.0000.00I-1".EPL_FB_OUT_136_I2008_S89Out;
	Cyclic#1.::gCommOutput.Array[137] AT %QW."8FLM01.0000.00I-1".EPL_FB_OUT_137_I2008_S8AOut;
	Cyclic#1.::gCommOutput.Array[138] AT %QW."8FLM01.0000.00I-1".EPL_FB_OUT_138_I2008_S8BOut;
	Cyclic#1.::gCommOutput.Array[139] AT %QW."8FLM01.0000.00I-1".EPL_FB_OUT_139_I2008_S8COut;
	Cyclic#1.::gCommOutput.Array[140] AT %QW."8FLM01.0000.00I-1".EPL_FB_OUT_140_I2008_S8DOut;
	Cyclic#1.::gCommOutput.Array[141] AT %QW."8FLM01.0000.00I-1".EPL_FB_OUT_141_I2008_S8EOut;
	Cyclic#1.::gCommOutput.Array[142] AT %QW."8FLM01.0000.00I-1".EPL_FB_OUT_142_I2008_S8FOut;
	Cyclic#1.::gCommOutput.Array[143] AT %QW."8FLM01.0000.00I-1".EPL_FB_OUT_143_I2008_S90Out;
	Cyclic#1.::gCommOutput.Array[144] AT %QW."8FLM01.0000.00I-1".EPL_FB_OUT_144_I2008_S91Out;
	Cyclic#1.::gCommOutput.Array[145] AT %QW."8FLM01.0000.00I-1".EPL_FB_OUT_145_I2008_S92Out;
	Cyclic#1.::gCommOutput.Array[146] AT %QW."8FLM01.0000.00I-1".EPL_FB_OUT_146_I2008_S93Out;
	Cyclic#1.::gCommOutput.Array[147] AT %QW."8FLM01.0000.00I-1".EPL_FB_OUT_147_I2008_S94Out;
	Cyclic#1.::gCommOutput.Array[148] AT %QW."8FLM01.0000.00I-1".EPL_FB_OUT_148_I2008_S95Out;
	Cyclic#1.::gCommOutput.Array[149] AT %QW."8FLM01.0000.00I-1".EPL_FB_OUT_149_I2008_S96Out;
	Cyclic#1.::gCommOutput.Array[150] AT %QW."8FLM01.0000.00I-1".EPL_FB_OUT_150_I2008_S97Out;
	Cyclic#1.::gCommOutput.Array[151] AT %QW."8FLM01.0000.00I-1".EPL_FB_OUT_151_I2008_S98Out;
	Cyclic#1.::gCommOutput.Array[152] AT %QW."8FLM01.0000.00I-1".EPL_FB_OUT_152_I2008_S99Out;
	Cyclic#1.::gCommOutput.Array[153] AT %QW."8FLM01.0000.00I-1".EPL_FB_OUT_153_I2008_S9AOut;
	Cyclic#1.::gCommOutput.Array[154] AT %QW."8FLM01.0000.00I-1".EPL_FB_OUT_154_I2008_S9BOut;
	Cyclic#1.::gCommOutput.Array[155] AT %QW."8FLM01.0000.00I-1".EPL_FB_OUT_155_I2008_S9COut;
	Cyclic#1.::gCommOutput.Array[156] AT %QW."8FLM01.0000.00I-1".EPL_FB_OUT_156_I2008_S9DOut;
	Cyclic#1.::gCommOutput.Array[157] AT %QW."8FLM01.0000.00I-1".EPL_FB_OUT_157_I2008_S9EOut;
	Cyclic#1.::gCommOutput.Array[158] AT %QW."8FLM01.0000.00I-1".EPL_FB_OUT_158_I2008_S9FOut;
	Cyclic#1.::gCommOutput.Array[159] AT %QW."8FLM01.0000.00I-1".EPL_FB_OUT_159_I2008_SA0Out;
	Cyclic#1.::gCommOutput.Array[160] AT %QW."8FLM01.0000.00I-1".EPL_FB_OUT_160_I2008_SA1Out;
	Cyclic#1.::gCommOutput.Array[161] AT %QW."8FLM01.0000.00I-1".EPL_FB_OUT_161_I2008_SA2Out;
	Cyclic#1.::gCommOutput.Array[162] AT %QW."8FLM01.0000.00I-1".EPL_FB_OUT_162_I2008_SA3Out;
	Cyclic#1.::gCommOutput.Array[163] AT %QW."8FLM01.0000.00I-1".EPL_FB_OUT_163_I2008_SA4Out;
	Cyclic#1.::gCommOutput.Array[164] AT %QW."8FLM01.0000.00I-1".EPL_FB_OUT_164_I2008_SA5Out;
	Cyclic#1.::gCommOutput.Array[165] AT %QW."8FLM01.0000.00I-1".EPL_FB_OUT_165_I2008_SA6Out;
	Cyclic#1.::gCommOutput.Array[166] AT %QW."8FLM01.0000.00I-1".EPL_FB_OUT_166_I2008_SA7Out;
	Cyclic#1.::gCommOutput.Array[167] AT %QW."8FLM01.0000.00I-1".EPL_FB_OUT_167_I2008_SA8Out;
	Cyclic#1.::gCommOutput.Array[168] AT %QW."8FLM01.0000.00I-1".EPL_FB_OUT_168_I2008_SA9Out;
	Cyclic#1.::gCommOutput.Array[169] AT %QW."8FLM01.0000.00I-1".EPL_FB_OUT_169_I2008_SAAOut;
	Cyclic#1.::gCommOutput.Array[170] AT %QW."8FLM01.0000.00I-1".EPL_FB_OUT_170_I2008_SABOut;
	Cyclic#1.::gCommOutput.Array[171] AT %QW."8FLM01.0000.00I-1".EPL_FB_OUT_171_I2008_SACOut;
	Cyclic#1.::gCommOutput.Array[172] AT %QW."8FLM01.0000.00I-1".EPL_FB_OUT_172_I2008_SADOut;
	Cyclic#1.::gCommOutput.Array[173] AT %QW."8FLM01.0000.00I-1".EPL_FB_OUT_173_I2008_SAEOut;
	Cyclic#1.::gCommOutput.Array[174] AT %QW."8FLM01.0000.00I-1".EPL_FB_OUT_174_I2008_SAFOut;
	Cyclic#1.::gCommOutput.Array[175] AT %QW."8FLM01.0000.00I-1".EPL_FB_OUT_175_I2008_SB0Out;
	Cyclic#1.::gCommOutput.Array[176] AT %QW."8FLM01.0000.00I-1".EPL_FB_OUT_176_I2008_SB1Out;
	Cyclic#1.::gCommOutput.Array[177] AT %QW."8FLM01.0000.00I-1".EPL_FB_OUT_177_I2008_SB2Out;
	Cyclic#1.::gCommOutput.Array[178] AT %QW."8FLM01.0000.00I-1".EPL_FB_OUT_178_I2008_SB3Out;
	Cyclic#1.::gCommOutput.Array[179] AT %QW."8FLM01.0000.00I-1".EPL_FB_OUT_179_I2008_SB4Out;
	Cyclic#1.::gCommOutput.Array[180] AT %QW."8FLM01.0000.00I-1".EPL_FB_OUT_180_I2008_SB5Out;
	Cyclic#1.::gCommOutput.Array[181] AT %QW."8FLM01.0000.00I-1".EPL_FB_OUT_181_I2008_SB6Out;
	Cyclic#1.::gCommOutput.Array[182] AT %QW."8FLM01.0000.00I-1".EPL_FB_OUT_182_I2008_SB7Out;
	Cyclic#1.::gCommOutput.Array[183] AT %QW."8FLM01.0000.00I-1".EPL_FB_OUT_183_I2008_SB8Out;
	Cyclic#1.::gCommOutput.Array[184] AT %QW."8FLM01.0000.00I-1".EPL_FB_OUT_184_I2008_SB9Out;
	Cyclic#1.::gCommOutput.Array[185] AT %QW."8FLM01.0000.00I-1".EPL_FB_OUT_185_I2008_SBAOut;
	Cyclic#1.::gCommOutput.Array[186] AT %QW."8FLM01.0000.00I-1".EPL_FB_OUT_186_I2008_SBBOut;
	Cyclic#1.::gCommOutput.Array[187] AT %QW."8FLM01.0000.00I-1".EPL_FB_OUT_187_I2008_SBCOut;
	Cyclic#1.::gCommOutput.Array[188] AT %QW."8FLM01.0000.00I-1".EPL_FB_OUT_188_I2008_SBDOut;
	Cyclic#1.::gCommOutput.Array[189] AT %QW."8FLM01.0000.00I-1".EPL_FB_OUT_189_I2008_SBEOut;
	Cyclic#1.::gCommOutput.Array[190] AT %QW."8FLM01.0000.00I-1".EPL_FB_OUT_190_I2008_SBFOut;
	Cyclic#1.::gCommOutput.Array[191] AT %QW."8FLM01.0000.00I-1".EPL_FB_OUT_191_I2008_SC0Out;
	Cyclic#1.::gCommOutput.Array[192] AT %QW."8FLM01.0000.00I-1".EPL_FB_OUT_192_I2008_SC1Out;
	Cyclic#1.::gCommOutput.Array[193] AT %QW."8FLM01.0000.00I-1".EPL_FB_OUT_193_I2008_SC2Out;
	Cyclic#1.::gCommOutput.Array[194] AT %QW."8FLM01.0000.00I-1".EPL_FB_OUT_194_I2008_SC3Out;
	Cyclic#1.::gCommOutput.Array[195] AT %QW."8FLM01.0000.00I-1".EPL_FB_OUT_195_I2008_SC4Out;
	Cyclic#1.::gCommOutput.Array[196] AT %QW."8FLM01.0000.00I-1".EPL_FB_OUT_196_I2008_SC5Out;
	Cyclic#1.::gCommOutput.Array[197] AT %QW."8FLM01.0000.00I-1".EPL_FB_OUT_197_I2008_SC6Out;
	Cyclic#1.::gCommOutput.Array[198] AT %QW."8FLM01.0000.00I-1".EPL_FB_OUT_198_I2008_SC7Out;
	Cyclic#1.::gCommOutput.Array[199] AT %QW."8FLM01.0000.00I-1".EPL_FB_OUT_199_I2008_SC8Out;

END_VAR
```

## Logical view

Binary libraries used (declarations not repeated): operator, runtime, AsIecCon, astime, AsZip, FileIO, AsBrMath, AsBrStr, brsystem, AsIODiag, sys_lib, AsTCP, standard, MpBase 6.6.0, McAcp6D 3.6.0, McBase 6.6.1, MpTraffic 3.6.0, SfDomain 6.0.0

### Global.typ - Global data types
```iecst
TYPE
	TaskDiagType : 	STRUCT
		Main : TaskEmStateInfoType;
		Power : TaskCmStateInfoType;
		FastDemo : TaskEmStateInfoType;
	END_STRUCT;
	TaskEmStateInfoType : 	STRUCT
		StateInfo : STRING[255];
		State : EMPackMLStateEnum;
		SubState : DINT;
		Mode : EMPackMLModeEnum;
		StateComplete : BOOL;
		WaitingForTask : STRING[255];
		Error : GeneralErrorInfoType;
	END_STRUCT;
	TaskCmStateInfoType : 	STRUCT
		StateInfo : STRING[255];
		State : DINT;
		SubState : DINT;
		Error : GeneralErrorInfoType;
	END_STRUCT;
	GeneralErrorInfoType : 	STRUCT
		Code : DINT;
		Description : STRING[80];
		AdditionalInfo : STRING[80];
		State : DINT;
		SubState : DINT;
	END_STRUCT;
END_TYPE

(**)

TYPE
	ShuttleListType : 	STRUCT
		Count : UDINT;
		Shuttle : ARRAY[0..gMAX_INDEX_SHUTTLE]OF ShuttleType;
	END_STRUCT;
	ShuttleType : 	STRUCT
		ID : UINT;
		UID : ShuttleUidType;
		Ref : Mc6DShuttleType;
		Position : McAcp6DShPositionType;
		MotionBuffer : McAcp6DShInfoMotionBufferType;
		State : McAcp6DShStateEnum;
	END_STRUCT;
	ShuttleUidType : 	STRUCT
		High : UDINT;
		Low : UDINT;
	END_STRUCT;
END_TYPE

(**)

TYPE
	DigitalInputs : 	STRUCT
		Button1 : BOOL;
		Button2 : BOOL;
		Button3 : BOOL;
	END_STRUCT;
	DigitalOutputs : 	STRUCT
		Button1_Led : BOOL;
		Button2_Led : BOOL;
		Button3_Led : BOOL;
	END_STRUCT;
END_TYPE
```

### Global.var - Global variables
```iecst
VAR CONSTANT
	gMAX_SHUTTLE_COUNT : UINT := 35; (*Maximum numer of shuttles on the system*)
	gMAX_INDEX_SHUTTLE : UINT := gMAX_SHUTTLE_COUNT-1; (*Maximum index for a shuttles on the system*)
END_VAR
(**)
(*6D Defaults*)
VAR CONSTANT
	gDEFAULT_Z : REAL := 0.0012;
END_VAR
(**)
(*6D Communication inteface*)
VAR
	gCommInput : Mc6DControllerFBIOType; (*Communication variable INPUT*)
	gCommOutput : Mc6DControllerFBIOType; (*Communication variable OUTPUT*)
END_VAR
(**)
(*Shuttles*)
VAR
	gShuttles : ShuttleListType;
END_VAR
(**)
(*PackML diagnostics*)
VAR
	gTasks : TaskDiagType;
END_VAR
(**)
(*IO*)
VAR
	gDI : DigitalInputs;
	gDO : DigitalOutputs;
END_VAR
```

### Package Logical/Libraries - Global libraries

### Library Logical/Libraries/SegFind (IEC)

#### SegFind.fun - Exported functions and function blocks
```iecst
FUNCTION_BLOCK Positioner
	VAR_INPUT
		Position : McAcp6DShPositionType;
	END_VAR
	VAR_OUTPUT
		Segment : USINT;
	END_VAR
	VAR
		X_Pos : REAL;
		Y_Pos : REAL;
		Row : USINT;
		Column : USINT;
	END_VAR
	VAR_INPUT
		Execute : BOOL;
	END_VAR
	VAR_OUTPUT
		Done : BOOL;
	END_VAR
END_FUNCTION_BLOCK
```

#### SegFind.st
```iecst
FUNCTION_BLOCK Positioner
	// We are not done
	Done := FALSE;

	// Get position
	X_Pos := Position.X;
	Y_Pos := Position.Y;

	// Then the position in segments
	Column := REAL_TO_USINT(brmceil(X_Pos / 0.24));
	Row := REAL_TO_USINT(brmceil(Y_Pos / 0.24));

	// Default
	Segment := 0;

	// Then we need to figure out which segment it is (welcome to switch-case -hell)
	CASE Column OF
		1:
			CASE Row OF
				1:
					Segment := 1;
				2:
					Segment := 2;
				7:
					Segment := 3;
				8:
					Segment := 4;
				13:
					Segment := 5;
				14:
					Segment := 6;
				19:
					Segment := 7;
				20:
					Segment := 8;

			END_CASE;
		2:
			Segment := 8 + Row;
		3:
			Segment := 28 + Row;
		4:
			CASE Row OF
				1:
					Segment := 49;
				2:
					Segment := 50;
				7:
					Segment := 51;
				8:
					Segment := 52;
				13:
					Segment := 53;
				14:
					Segment := 54;
				19:
					Segment := 55;
				20:
					Segment := 56;

			END_CASE;
	END_CASE;

	// Now we are
	Done := TRUE;
END_FUNCTION_BLOCK
```

### Library Logical/Libraries/Mover (IEC)

#### Types.typ - Exported data types
```iecst
TYPE
	MoveCommandType : 	STRUCT  (*Contains an X and a Y in REAL*)
		X : REAL;
		Y : REAL;
	END_STRUCT;
END_TYPE
```

#### Mover.fun - Exported functions and function blocks
```iecst
FUNCTION_BLOCK QuarterMover
	VAR_INPUT
		Position : McAcp6DShPositionType;
		SegmentPosition : MoveCommandType;
		Execute : BOOL;
	END_VAR
	VAR
		XDiff : REAL;
		YDiff : REAL;
	END_VAR
	VAR_OUTPUT
		MoveCommand : MoveCommandType;
		Done : BOOL;
	END_VAR
END_FUNCTION_BLOCK

FUNCTION_BLOCK CenterMover
	VAR_INPUT
		Segment : USINT;
		Execute : BOOL;
	END_VAR
	VAR_OUTPUT
		MoveCommand : MoveCommandType;
		Done : BOOL;
	END_VAR
END_FUNCTION_BLOCK

FUNCTION_BLOCK Mover
	VAR_INPUT
		Segment : USINT;
		Execute : BOOL;
	END_VAR
	VAR_OUTPUT
		MoveCommand : MoveCommandType;
		Done : BOOL;
	END_VAR
END_FUNCTION_BLOCK
```

#### Mover.st
```iecst
FUNCTION_BLOCK Mover
	// We are not done
	Done := FALSE;

	// Initialize, so we don't have empty values
	MoveCommand.X := 0;
	MoveCommand.Y := 0;

	// Let's try stuff
	IF Segment = 1 THEN
		MoveCommand.X := 0.72;
		MoveCommand.Y := 0;
	ELSIF Segment <= 8 THEN
		MoveCommand.X := 0.24 * (Segment MOD 2);
		MoveCommand.Y := -0.24 * (1 - (Segment MOD 2));
	ELSIF (Segment = 10) OR (Segment = 16) OR (Segment = 22) THEN
		MoveCommand.X := -0.24;
		MoveCommand.Y := 0;
	ELSIF (Segment >= 11) AND (Segment <= 27) THEN
		MoveCommand.X := 0;
		MoveCommand.Y := 0.24*(5 - ((Segment - 6*REAL_TO_USINT(brmceil((Segment - 3)/6))+2) MOD 6)) - 1.2;
	ELSIF (Segment = 35) OR (Segment = 41) OR (Segment = 47) THEN
		MoveCommand.X := 0.24;
		MoveCommand.Y := 0;
	ELSIF (Segment >= 30) AND (Segment <= 46) THEN
		MoveCommand.X := 0;
		MoveCommand.Y := 1.2 - 0.24*((Segment - 6*REAL_TO_USINT(brmceil((Segment - 3)/6))) MOD 6);
	ELSIF (Segment >= 49) AND (Segment <= 55) THEN
		MoveCommand.X := -0.24 * (1 - (Segment MOD 2));
		MoveCommand.Y := 0.24 * (Segment MOD 2);
	ELSIF Segment = 56 THEN
		MoveCommand.X := -0.72;
		MoveCommand.Y := 0;
	ELSIF Segment = 9 THEN    // Everything after this is just ductape and dreams
		MoveCommand.X := 0.48;
		MoveCommand.Y := 0;
	ELSIF Segment = 29 THEN
		MoveCommand.X := 0.24;
		MoveCommand.Y := 0;
	ELSIF Segment = 28 THEN
		MoveCommand.X := -0.24;
		MoveCommand.Y := 0;
	ELSIF Segment = 48 THEN
		MoveCommand.X := -0.48;
		MoveCommand.Y := 0;
	END_IF;

	// Now we are
	Done := TRUE;
END_FUNCTION_BLOCK
```

#### CenterMover.st
```iecst
FUNCTION_BLOCK CenterMover
	// We are not done
	Done := FALSE;

	// Initialize, so we don't have empty values
	MoveCommand.X := 0;
	MoveCommand.Y := 0;

	// Once again, welcome to if-else -hell
	IF Segment >= 1 AND Segment <= 8 THEN
		MoveCommand.X := 120;
		CASE Segment OF
			1:
				MoveCommand.Y := 120;
			2:
				MoveCommand.Y := 360;
			3:
				MoveCommand.Y := 1560;
			4:
				MoveCommand.Y := 1800;
			5:
				MoveCommand.Y := 3000;
			6:
				MoveCommand.Y := 3240;
			7:
				MoveCommand.Y := 4440;
			8:
				MoveCommand.Y := 4680;
		END_CASE;
	ELSIF Segment <= 28 THEN
		MoveCommand.X := 360;
		MoveCommand.Y := 240*(Segment-9) + 120;
	ELSIF Segment <= 48 THEN
		MoveCommand.X := 600;
		MoveCommand.Y := 240*(Segment-29) + 120;
	ELSIF Segment >= 49 THEN
		MoveCommand.X := 840;
		CASE Segment OF
			49:
				MoveCommand.Y := 120;
			50:
				MoveCommand.Y := 360;
			51:
				MoveCommand.Y := 1560;
			52:
				MoveCommand.Y := 1800;
			53:
				MoveCommand.Y := 3000;
			54:
				MoveCommand.Y := 3240;
			55:
				MoveCommand.Y := 4440;
			56:
				MoveCommand.Y := 4680;
		END_CASE;
	END_IF;

	// I forgot that these are in meters, not millimeters :))))
	MoveCommand.X := MoveCommand.X / 1000;
	MoveCommand.Y := MoveCommand.Y / 1000;

	// Now we are
	Done := TRUE;
	END_FUNCTION_BLOCK
```

#### QuarterMover.st
```iecst
FUNCTION_BLOCK QuarterMover
	// We are not done
	Done := FALSE;

	// Initialize, so we don't have empty values
	MoveCommand.X := SegmentPosition.X;
	MoveCommand.Y := SegmentPosition.Y;

	// Let's determine where in relation to the center the segment is
	XDiff := Position.X - SegmentPosition.X;
	YDiff := Position.Y - SegmentPosition.Y;

	// Then the good old if-else -hell :)
	IF (XDiff < 0) AND (YDiff < 0) THEN
		MoveCommand.X := MoveCommand.X - 0.06;
		MoveCommand.Y := MoveCommand.Y - 0.06;
	ELSIF (XDiff < 0) AND (YDiff > 0) THEN
		MoveCommand.X := MoveCommand.X - 0.06;
		MoveCommand.Y := MoveCommand.Y + 0.06;
	ELSIF (XDiff > 0) AND (YDiff < 0) THEN
		MoveCommand.X := MoveCommand.X + 0.06;
		MoveCommand.Y := MoveCommand.Y - 0.06;
	ELSIF (XDiff > 0) AND (YDiff > 0) THEN
		MoveCommand.X := MoveCommand.X + 0.06;
		MoveCommand.Y := MoveCommand.Y + 0.06;
	END_IF;

	// Now we are
	Done := TRUE;
	END_FUNCTION_BLOCK
```

### Library Logical/Libraries/BrdkPackML (ANSIC, version 2.0.0) - OMAC PackML
Depends on: sys_lib, brsystem

#### BrdkPackML.fun
```iecst
FUNCTION_BLOCK ControlModule (*Control module implementation for OMAC PackML*)
	VAR_INPUT
		Setup : CMSetupType; (*Local setup*) (* *) (*#PAR#;*)
		Interface : CMInterfaceType; (*Publish/Subscribe Interface between Equipment Modules *)
		StateInfo : STRING[255]; (*Status of what the substate is doing or waiting for. Will also be used for logging.*) (* *) (*#CYC#;*)
		State : DINT; (*Control Module state*)
		SubState : DINT := 0; (*The sub state of the module. Can be used for programming the sequence inside a PackML state. Will automatically be reset to 0 by a PackML state change.*) (* *) (*#CYC#;*)
	END_VAR
	VAR_OUTPUT
		Info : CMInfoType; (*Additional information about the component*) (* *) (*#CMD#; *)
	END_VAR
	VAR
		Internal : CMInternalType; (*Internal variables*)
	END_VAR
END_FUNCTION_BLOCK

FUNCTION_BLOCK EquipmentModule (*Synchronized PackML state machine handling*) (* $GROUP=mapp Services,$CAT=OMAC PackML,$GROUPICON=Icon_mapp.png,$CATICON=Icon_MpPackML.png *)
	VAR_INPUT
		Setup : EMSetupType; (*Local setup*) (* *) (*#PAR#;*)
		Interface : EMInterfaceType; (*Publish/Subscribe Interface between Equipment Modules *)
		SetModeID : DINT := 1; (*Change the packML mode*)
		StateInfo : STRING[255]; (*Status of what the substate is doing or waiting for. Will also be used for logging.*) (* *) (*#CYC#;*)
		Command : EMCommandType; (*Control commands from ISA-TR88.00.02 commands.*) (* *) (*#CMD#;*)
		SubState : DINT := 0; (*The sub state of the module. Can be used for programming the sequence inside a PackML state. Will automatically be reset to 0 by a PackML state change.*) (* *) (*#CYC#;*)
	END_VAR
	VAR_OUTPUT
		StateCurrent : EMPackMLStateEnum := STATE_UNDEFINED; (*Current state*) (* *) (*#CMD#;*)
		ModeID : EMPackMLModeEnum := MODE_PRODUCTION; (*The current mode*) (* *) (*#CMD#;*)
		Info : EMInfoType; (*Additional information about the component*) (* *) (*#CMD#; *)
	END_VAR
	VAR
		Internal : EMInternalType; (*Internal variables*)
	END_VAR
END_FUNCTION_BLOCK

FUNCTION EMGetModuleAdrByIdx : UDINT (*Returns the address of an Equipment Module on the heap based on the index*)
	VAR_INPUT
		EmIdx : UDINT; (*Index of the Equipment Module*)
	END_VAR
END_FUNCTION

FUNCTION EMGetModuleIdxByName : UDINT (*Returns the index for an Em with the specified name*)
	VAR_INPUT
		EmName : STRING[255]; (*Name of the Equipment Module*)
	END_VAR
END_FUNCTION

FUNCTION EMGetModuleAdrByName : UDINT (*Returns the address of an Equipment Module on the heap based on its name*)
	VAR_INPUT
		EmName : STRING[255]; (*Name of the Equipment Module*)
	END_VAR
END_FUNCTION

FUNCTION EMGetNumberOfModules : UDINT (*Returns the number of Equipment Modules*)
END_FUNCTION

FUNCTION EMGetNumberOfRootModules : UDINT (*Returns the number of root modules. A root module is an Equipment Module with Level 0*)
END_FUNCTION

FUNCTION EMGetWaitingForByIdx : BOOL (*Get WaitingFor from hierarchy index. Returns true on success*)
	VAR_INPUT
		EmIdx : UDINT; (*Index of the root*)
		WaitingFor : EMStatusType; (*EMStatusType*)
	END_VAR
END_FUNCTION

FUNCTION EMGetInterruptedByByIdx : BOOL (*Get InterruptedBy from hierarchy index. Returns true on success*)
	VAR_INPUT
		EmIdx : UDINT; (*Index of the root*)
		InterruptedBy : EMStatusType; (*EMStatusType*)
	END_VAR
END_FUNCTION

FUNCTION EMGetModuleStatus : BOOL (*Get the status from any Equipment Module using the memory address. Returns true on success*)
	VAR_INPUT
		EmAddress : UDINT; (*Address of the Equipment Module*)
		EMStatus : EMStatusType; (*EMStatusType*)
	END_VAR
END_FUNCTION

FUNCTION EMGetModuleStatusByName : BOOL (*Get the status from any Equipment Module using the configured name. Returns true on success*)
	VAR_INPUT
		EmName : STRING[255]; (*Name of the Equipment Module*)
		EMStatus : EMStatusType; (*EMStatusType*)
	END_VAR
END_FUNCTION

FUNCTION EMGetModuleStatusByIdx : BOOL (*Get the status from any Equipment Module using an index. Returns true on success*)
	VAR_INPUT
		EmIdx : UDINT; (*Index of the Equipment Module*)
		EMStatus : EMStatusType; (*EMStatusType*)
	END_VAR
END_FUNCTION

FUNCTION EMGetParentAdr : UDINT (*Returns the address of the parent Equipment Module on the heap*)
	VAR_INPUT
		EmAddress : UDINT; (*Address of the Equipment Module*)
	END_VAR
END_FUNCTION

FUNCTION EMGetChildrenAdrByIdx : UDINT (*Returns the address of a child Equipment Module using an index*)
	VAR_INPUT
		EmAddress : UDINT; (*Address of the Equipment Module*)
		EmIdx : UDINT; (*Index of the child Equipment Module*)
	END_VAR
END_FUNCTION

FUNCTION EMGetSiblingAdrByIdx : UDINT (*Returns the address of a sibling Equipment Module using an index*)
	VAR_INPUT
		EmAddress : UDINT; (*Address of the Equipment Module*)
		EmIdx : UDINT; (*Index of the sibling Equipment Module*)
	END_VAR
END_FUNCTION

FUNCTION EMGetRootAdrByIdx : UDINT (*Returns the address of a root Equipment Module using an index*)
	VAR_INPUT
		EmIdx : UDINT; (*Index of a root Equipment Module*)
	END_VAR
END_FUNCTION

FUNCTION EMGetUserDataAdr : UDINT (*Returns the address of the published userdata from a remote Equipment Module*)
	VAR_INPUT
		EmAddress : UDINT; (*Address of the Equipment Module*)
	END_VAR
END_FUNCTION

FUNCTION EMSetCommand : BOOL (*Send a command to an Equipment Module using its address. Returns true on success*)
	VAR_INPUT
		EmAddress : UDINT; (*Address of the remote Equipment Module to receive the command*)
		EmAddressInterrupter : UDINT; (*Address of the local Equipment Module interrupting the remote Em *)
		Command : EMPackMLCmdEnum; (*Command*)
	END_VAR
END_FUNCTION

FUNCTION EMSetMode : BOOL (*Function changing the mode of an Equipment Module*) (* $GROUP=mapp Services,$CAT=OMAC PackML,$GROUPICON=Icon_mapp.png,$CATICON=Icon_MpPackML.png *)
	VAR_INPUT
		EmAddress : UDINT; (*Address of the target Equipment Module*)
		Mode : DINT; (*Desired mode to change to. The mode must be defined in the mppackmlcore configuration*) (* *) (*#PAR#;*)
	END_VAR
END_FUNCTION

FUNCTION EMSetModeByName : BOOL (*Function changing the mode of an Equipment Module*) (* $GROUP=mapp Services,$CAT=OMAC PackML,$GROUPICON=Icon_mapp.png,$CATICON=Icon_MpPackML.png *)
	VAR_INPUT
		EmName : STRING[255]; (*Name of the target Equipment Module*)
		Mode : DINT; (*Desired mode to change to. *) (* *) (*#PAR#;*)
	END_VAR
END_FUNCTION
```

#### BrdkPackML.typ
```iecst
TYPE
	EMStatusType : 	STRUCT  (*EMStatusType*)
		Name : STRING[255]; (*Em Name*)
		ModeID : UDINT; (*Current Mode*)
		StateCurrent : EMPackMLStateEnum; (*Current State*)
		SubStateCurrent : DINT; (*Current Sub State*)
		StateComplete : BOOL; (*State Complete*)
		StateInfo : STRING[255]; (*Used to describe the action in all states and substates*)
	END_STRUCT;
	EMCommandType : 	STRUCT  (*EMCommandType*)
		Abort : BOOL; (*Go to state Aborting - Can be set in all states except Aborting and Aborted.*)
		Clear : BOOL; (*Go to state Clearing - Can only be set in state Aborted.*)
		Stop : BOOL; (*Go to state Stopping - Can be set in all states except Aborting, Aborted, Clearing, Stopping and Stopped.*)
		Reset : BOOL; (*Go to state Resetting - Can only be set in state Stopped.*)
		Start : BOOL; (*Go to state Starting - Can only be set in state Idle.*)
		Hold : BOOL; (*Go to state Holding. Can only be set in state Execute.*)
		Unhold : BOOL; (*Go to state Unholding. Can only be set in state Held.*)
		Suspend : BOOL; (*Go to state Suspending. Can only be set in state Execute.*)
		Unsuspend : BOOL; (*Go to state Unsuspending. Can only be set in state Suspended.*)
		Complete : BOOL; (*Go to state Completing. Can only be set in state Execute*)
		StateComplete : BOOL; (*Go to next waiting state. Can be set in all acting states and state Execute.*)
	END_STRUCT;
	EMPackMLCmdEnum :
		( (*Command Enum*)
		CMD_UNDEFINED := 0, (*Undefined Command*)
		CMD_RESET := 1, (*PackML Reset Command*)
		CMD_START := 2, (*PackML Start Command*)
		CMD_STOP := 3, (*PackML Stop Command*)
		CMD_HOLD := 4, (*PackML Hold Command*)
		CMD_UNHOLD := 5, (*PackML Unhold Command*)
		CMD_SUSPEND := 6, (*PackML Suspend Command*)
		CMD_UNSUSPEND := 7, (*PackML Unsuspend Command*)
		CMD_ABORT := 8, (*PackML Abort Command*)
		CMD_CLEAR := 9, (*PackML Clear Command*)
		CMD_COMPLETE := 10, (*PackML Complete Command*)
		CMD_SC := 11 (*PackML State Complete Command*)
		);
	EMPackMLModeEnum :
		( (*Mode Enum*)
		MODE_UNDEFINED := 0, (*PackML Undefined mode*)
		MODE_PRODUCTION := 1, (*PackML Production mode*)
		MODE_MAINTENANCE := 2, (*PackML Maintenance mode*)
		MODE_MANUAL := 3, (*PackML Manual mode*)
		MODE_CLEAN := 16, (*PackML Cleaning mode*)
		MODE_JOG := 17, (*PackML Jogging mode*)
		MODE_CIP := 18, (*PackML CIP mode*)
		MODE_CALIBRATION := 19 (*PackML Calibration mode*)
		);
	EMPackMLStateEnum :
		( (*State Enum*)
		STATE_UNDEFINED := 0, (*The system is inactive, no state active*)
		STATE_CLEARING := 1, (*PackML CLEARING state*)
		STATE_STOPPED := 2, (*PackML STOPPED state*)
		STATE_STARTING := 3, (*PackML STARTING state*)
		STATE_IDLE := 4, (*PackML IDLE state*)
		STATE_SUSPENDED := 5, (*PackML SUSPENDED state*)
		STATE_EXECUTE := 6, (*PackML EXECUTE state*)
		STATE_STOPPING := 7, (*PackML STOPPING state*)
		STATE_ABORTING := 8, (*PackML ABORTING state*)
		STATE_ABORTED := 9, (*PackML ABORTED state*)
		STATE_HOLDING := 10, (*PackML HOLDING state*)
		STATE_HELD := 11, (*PackML HELD state*)
		STATE_UNHOLDING := 12, (*PackML UNHOLDING state*)
		STATE_SUSPENDING := 13, (*PackML SUSPENDING state*)
		STATE_UNSUSPENDING := 14, (*PackML UNSUSPENDING state*)
		STATE_RESETTING := 15, (*PackML RESETTING state*)
		STATE_COMPLETING := 16, (*PackML COMPLETING state*)
		STATE_COMPLETED := 17, (*PackML COMPLETED state*)
		STATE_DEACTIVATING := 30, (*Deactivating state. Not a standard PackML state*)
		STATE_DEACTIVATED := 31, (*Deactivated state. Not a standard PackML state*)
		STATE_ACTIVATING := 32 (*Activating state. Not a standard PackML state*)
		);
	EMActivationConditionEnum :
		( (*Activation Enum*)
		ACTIVATE_AUTOMATIC := 0, (*Activate Em automatically when executed*)
		ACTIVATE_BY_PARENT := 1, (*Activate Em if parent is activated*)
		ACTIVATE_BY_PV := 2 (*Activate Em based on PV value*)
		);
	EMSetupType : 	STRUCT  (*EMSetupType*)
		ParentName : STRING[255]; (*Name of the parent. Leave empty is Em is parent at level 0*)
		Name : STRING[255]; (*Name of the Em. If left empty during first execution, the task name is used as Em name*)
		NameIndex : USINT := EM_MAX_NAME_INDEX; (*Index of the Em if having multiple Em's in an array*)
		Activate : BOOL := FALSE; (*PV for ActivationCondition ACTIVATE_BY_PV*)
		ActivationCondition : EMActivationConditionEnum := ACTIVATE_AUTOMATIC; (*Condition for activating the Em*)
		EnableWaitingFor : BOOL := TRUE; (*Enable the WaitingFor log*)
		EnableInteruptedBy : BOOL := TRUE; (*Enable the InterruptedBy log*)
		Synchronisation : EMSynchronisationType; (*Parameters for Em synchronization*)
		AuditModeChange : BOOL := TRUE; (*Log when mode is changed*)
		AuditStateChange : BOOL := TRUE; (*Log when state is changed*)
		AuditSubStateChange : BOOL := TRUE; (*Log when substate is changed*)
		SkipStopStateComplete : BOOL; (*The StateComplete command is ignored during stop*)
	END_STRUCT;
	EMInfoType : 	STRUCT  (*EMInfoType*)
		ParentName : STRING[255]; (*Name of the Parent Em*)
		ParentStateCurrent : EMPackMLStateEnum; (*Parent Current State*)
		EmName : STRING[255]; (*Name of the Em*)
		EmAddress : UDINT; (*Address of the Em*)
		EmIndex : UDINT; (*Global EM index*)
		UserDataAddress : UDINT; (*Published data address*)
		Level : UDINT; (*Level in the hierarchy. Parent is level 0.*)
		SiblingCount : UDINT; (*Number of Siblings. No siblings means Sibling count 1*)
		ChildCount : UDINT; (*How many children are registered to this module. Even when desynchronised the child count will still be valid.*)
		ParentStateComplete : BOOL; (*The parent is state complete. Can be used to synchronize a state transition*)
		SiblingsStateComplete : BOOL; (*All siblings are state complete. Can be used to synchronize a state transition*)
		ChildrenStateComplete : BOOL; (*All children are state complete. Can be used to synchronize a state transition*)
		WaitingFor : EMStatusType; (*The status for the Em we are waiting for*)
		InteruptedBy : EMStatusType; (*The Em we where interrupted by*)
		TimeInState : REAL; (*The actual time in the current state*)
		TimeInSubState : REAL; (*The actual time in the current sub state*)
		Last : ARRAY[0..EM_MAX_AUDIT_ENTRIES]OF STRING[50]; (*The last state, substate and mode*)
		CycleTime : REAL; (*Cycle Time in seconds*)
		OnStateEntry : BOOL; (*Goes to true on the first scan after a state change*)
		OnSubStateEntry : BOOL; (*Goes to true on the first scan after a substate change*)
	END_STRUCT;
	EMInternalType : 	STRUCT  (*Internal type of the Em*)
		state : USINT; (*Internal state*)
		emAddress : UDINT; (*Address of the instance on the heap memory*)
		userDataAddress : UDINT; (*Address of the user data on the heap memory*)
		subscriptionUserDataAddress : ARRAY[0..EM_MAX_SUBSCRIPTIONS]OF UDINT; (*Address of the user data we are currently subscribing to*)
		subscribedToEMName : ARRAY[0..EM_MAX_SUBSCRIPTIONS]OF STRING[255]; (*Name of the Em we are subscribed to*)
		oldPubSubEnable : BOOL; (*Old Pub/Sub enable*)
	END_STRUCT;
	EMSynchronisationType : 	STRUCT  (*Em synchronization settings type*)
		Override : EMSynchronisationCmdType := (Abort:=FALSE,Stop:=FALSE,Complete:=FALSE,Suspend:=FALSE,Unsuspend:=FALSE,Hold:=FALSE,Unhold:=TRUE,Clear:=TRUE,Reset:=TRUE,Start:=TRUE); (*Commands that are overriden by parrent command*)
		ReactTo : EMSynchronisationCmdType := (Abort:=TRUE,Stop:=TRUE,Complete:=TRUE,Suspend:=TRUE,Unsuspend:=TRUE,Hold:=TRUE,Unhold:=TRUE,Clear:=TRUE,Reset:=TRUE,Start:=TRUE); (*Commands that are reacted to by parent*)
		Escalate : EMSynchronisationCmdType := (Abort:=TRUE,Stop:=TRUE,Complete:=TRUE,Suspend:=TRUE,Unsuspend:=TRUE,Hold:=TRUE,Unhold:=FALSE,Clear:=FALSE,Reset:=FALSE,Start:=FALSE); (*Commands that are escalated to the parrent*)
	END_STRUCT;
	EMSynchronisationCmdType : 	STRUCT  (*Em synchronization settings type*)
		Abort : BOOL := FALSE; (*Synchronization setting for command*)
		Stop : BOOL := FALSE; (*Synchronization setting for command*)
		Complete : BOOL := FALSE; (*Synchronization setting for command*)
		Suspend : BOOL := FALSE; (*Synchronization setting for command*)
		Unsuspend : BOOL := FALSE; (*Synchronization setting for command*)
		Hold : BOOL := FALSE; (*Synchronization setting for command*)
		Unhold : BOOL := FALSE; (*Synchronization setting for command*)
		Clear : BOOL := FALSE; (*Synchronization setting for command*)
		Reset : BOOL := FALSE; (*Synchronization setting for command*)
		Start : BOOL := FALSE; (*Synchronization setting for command*)
	END_STRUCT;
	EMInterfaceType : 	STRUCT  (*Interface type*)
		Enable : BOOL; (*Enable Pub/Sub interface*)
		SubscriptionEMName : ARRAY[0..EM_MAX_SUBSCRIPTIONS]OF STRING[255]; (*Name of the Em where we want cyclic user data from*)
		SubscriptionValid : ARRAY[0..EM_MAX_SUBSCRIPTIONS]OF BOOL; (*True if data is valid. Only true if Em name does exist*)
		Publish : EMUserDataPubSubType; (*The local user data that other Em can subscribe to*)
		Subscribe : ARRAY[0..EM_MAX_SUBSCRIPTIONS]OF EMUserDataPubSubType; (*The user data from the remote Em that we are subscribing to*)
	END_STRUCT;
END_TYPE

(*CM*)

TYPE
	CMInternalType : 	STRUCT  (*Internal type of the Cm*)
		state : USINT; (*Internal state*)
		parentEmAddress : UDINT; (*Address of the instance on the heap memory*)
		subscriptionUserDataAddress : ARRAY[0..EM_MAX_SUBSCRIPTIONS]OF UDINT; (*Address of the user data we are currently subscribing to*)
		subscribedToEMName : ARRAY[0..EM_MAX_SUBSCRIPTIONS]OF STRING[255]; (*Name of the Em we are subscribed to*)
		oldState : DINT; (*Old state*)
		oldSubState : DINT; (*Old sub state*)
		cycleTime : REAL; (*Cycle time for the module task class*)
		oldPubSubEnable : BOOL; (*Old Pub/Sub enable*)
	END_STRUCT;
	CMSetupType : 	STRUCT  (*CMSetupType*)
		ParentName : STRING[255]; (*Name of the parent. Leave empty is Em is parent at level 0*)
		Name : STRING[255]; (*Name of the Em. If left empty during first execution, the task name is used as Em name*)
		NameIndex : USINT := EM_MAX_NAME_INDEX;
		AuditStateChange : BOOL := TRUE; (*Log when state is changed*)
		AuditSubStateChange : BOOL := TRUE; (*Log when substate is changed*)
	END_STRUCT;
	CMInfoType : 	STRUCT  (*CMInfoType*)
		CmName : STRING[255]; (*Name of the Cm*)
		ParentName : STRING[255]; (*Name of the Parent Em*)
		ParentEmAddress : UDINT; (*Address of the Em*)
		ParentEmIndex : UDINT; (*Global EM index*)
		ParentStateCurrent : EMPackMLStateEnum; (*Parent Current State*)
		Level : UDINT; (*Level in the hierarchy. Parent is level 0.*)
		TimeInState : REAL; (*The actual time in the current state*)
		TimeInSubState : REAL; (*The actual time in the current sub state*)
		Last : ARRAY[0..EM_MAX_AUDIT_ENTRIES]OF STRING[50]; (*The last state, substate and mode*)
		CycleTime : REAL; (*Cycle Time in seconds*)
		OnStateEntry : BOOL; (*True in first scan after a state change*)
		OnSubStateEntry : BOOL; (*True in first scan after a substate change*)
	END_STRUCT;
	CMInterfaceType : 	STRUCT  (*Interface type*)
		Enable : BOOL; (*Enable Sub interface*)
		SubscriptionEMName : ARRAY[0..EM_MAX_SUBSCRIPTIONS]OF STRING[255]; (*Name of the Em where we want cyclic user data from*)
		SubscriptionValid : ARRAY[0..EM_MAX_SUBSCRIPTIONS]OF BOOL; (*True if data is valid. Only true if Em name does exist*)
		Subscribe : ARRAY[0..EM_MAX_SUBSCRIPTIONS]OF EMUserDataPubSubType; (*The user data from the remote Em that we are subscribing to*)
	END_STRUCT;
END_TYPE

(******* USER DEFINED *******)

TYPE
	EMUserDataPubSubType : 	STRUCT  (*Local / Remote user data. This datatype can be expanded to fit the needs of the application*)
		State : EMPackMLStateEnum;
		SubState : DINT;
		StateComplete : BOOL;
		CmdAbortCounter : UDINT;
		CmdStopCounter : UDINT;
		Priority : UDINT;
		PrioritySC : BOOL;
	END_STRUCT;
END_TYPE
```

#### BrdkPackML.var
```iecst
VAR CONSTANT
	EM_MAX_NAME_INDEX : USINT := 255;
	EM_MAX_SUBSCRIPTIONS : USINT := 1; (*2*)
	EM_MAX_AUDIT_ENTRIES : USINT := 9; (*10*)
END_VAR
```

#### BrdkPackMLFunctions.cpp
```cpp
#include "BrdkPackML.h"
#include "../PackMLCore/PackMLModule.hpp"
#include "../PackMLCore/PackMLModuleTable.hpp"

unsigned long bur_heap_size = 0x3CCCC;

PackMLModuleTable* pPackMLModuleTable = new PackMLModuleTable();

//---------------------- IEC Functions ----------------------------------//
bool EMSetMode(unsigned long EmAddress, signed long Mode)
{
	if(EmAddress == 0){
		return false;
	}

	PackMLModule* pPackMLModule = reinterpret_cast<PackMLModule*>(EmAddress);

	return pPackMLModule->setCurrentMode(Mode);

}

bool EMSetModeByName(plcstring* EmName, signed long Mode)
{
	PackMLModule* pPackMLModule = pPackMLModuleTable->getModuleByName(EmName);

	if(pPackMLModule == nullptr)
		return false;

	return pPackMLModule->setCurrentMode(Mode);

}

plcbit EMGetModuleStatusByName(plcstring* EmName, struct EMStatusType* EMStatus){

	PackMLModule* pPackMLModule = pPackMLModuleTable->getModuleByName(EmName);

	if(EMStatus == 0 || pPackMLModule == nullptr){
		return false;
	}

	EMStatus->ModeID = pPackMLModule->getCurrentMode();
	strcpy(EMStatus->Name, pPackMLModule->getModuleName());
	EMStatus->StateComplete = pPackMLModule->getStateComplete();
	EMStatus->StateCurrent = static_cast<EMPackMLStateEnum>(pPackMLModule->getCurrentState());
	EMStatus->SubStateCurrent = pPackMLModule->getCurrentSubState();
	strcpy(EMStatus->StateInfo, pPackMLModule->getStateInfo());

	return true;
}

plcbit EMGetWaitingForByIdx(unsigned long EmIdx, struct EMStatusType* WaitingFor){
	PackMLModule* pPackMLModule = pPackMLModuleTable->getRootModuleByIdx(EmIdx);

	if(WaitingFor == 0 || pPackMLModule == nullptr){
		return false;
	}
	// Get waiting for info
	PackMLModuleSharedInfo* pWaitingFor =  pPackMLModule->getWaitingForPtr();
	if(pWaitingFor != nullptr){
		WaitingFor->ModeID = pWaitingFor->getModeCurrent();
		WaitingFor->StateCurrent = static_cast<EMPackMLStateEnum>(pWaitingFor->getStateCurrent());
		WaitingFor->SubStateCurrent = pWaitingFor->getSubStateCurrent();
		WaitingFor->StateComplete = pWaitingFor->getStateComplete();
		strcpy(WaitingFor->Name, pWaitingFor->getName());
		strcpy(WaitingFor->StateInfo, pWaitingFor->getStateInfo());
	} else {
		memset(&WaitingFor, 0, sizeof(WaitingFor));
	}
	return true;
}

plcbit EMGetInterruptedByByIdx(unsigned long EmIdx, struct EMStatusType* InterruptedBy){
	PackMLModule* pPackMLModule = pPackMLModuleTable->getRootModuleByIdx(EmIdx);

	if(InterruptedBy == 0 || pPackMLModule == nullptr){
		return false;
	}
	// Get interrupted by info
	PackMLModuleSharedInfo* pInteruptedBy =  pPackMLModule->getInteruptedByPtr();
	if(pInteruptedBy != nullptr){
		InterruptedBy->ModeID = pInteruptedBy->getModeCurrent();
		InterruptedBy->StateCurrent = static_cast<EMPackMLStateEnum>(pInteruptedBy->getStateCurrent());
		InterruptedBy->SubStateCurrent = pInteruptedBy->getSubStateCurrent();
		InterruptedBy->StateComplete = pInteruptedBy->getStateComplete();
		strcpy(InterruptedBy->Name, pInteruptedBy->getName());
		strcpy(InterruptedBy->StateInfo, pInteruptedBy->getStateInfo());
	} else {
		memset(&InterruptedBy, 0, sizeof(InterruptedBy));
	}
	return true;
}

unsigned long EMGetModuleAdrByName(plcstring* EmName){

	return reinterpret_cast<unsigned long int>(pPackMLModuleTable->getModuleByName(EmName));
}

unsigned long EMGetModuleAdrByIdx(unsigned long EmIdx){

	return reinterpret_cast<unsigned long int>(pPackMLModuleTable->getModuleByIdx(EmIdx));
}

plcbit EMGetModuleStatus(unsigned long EmAddress, struct EMStatusType* EMStatus){

	if(EmAddress == 0 || EMStatus == 0){
		return false;
	}

	PackMLModule* pPackMLModule = reinterpret_cast<PackMLModule*>(EmAddress);

	EMStatus->ModeID = pPackMLModule->getCurrentMode();
	strcpy(EMStatus->Name, pPackMLModule->getModuleName());
	EMStatus->StateComplete = pPackMLModule->getStateComplete();
	EMStatus->StateCurrent = static_cast<EMPackMLStateEnum>(pPackMLModule->getCurrentState());
	EMStatus->SubStateCurrent = pPackMLModule->getCurrentSubState();
	strcpy(EMStatus->StateInfo, pPackMLModule->getStateInfo());

	return true;
}

unsigned long EMGetNumberOfModules(){
	return pPackMLModuleTable->getNumberOfModules();
}

unsigned long EMGetNumberOfRootModules(){
	return pPackMLModuleTable->getNumberOfRoots();
}

plcbit EMGetModuleStatusByIdx(unsigned long EmIdx, struct EMStatusType* EMStatus){

	if(EMStatus == 0){
		return false;
	}

	PackMLModule* pPackMLModule = pPackMLModuleTable->getModuleByIdx(EmIdx);

	EMStatus->ModeID = pPackMLModule->getCurrentMode();
	strcpy(EMStatus->Name, pPackMLModule->getModuleName());
	EMStatus->StateComplete = pPackMLModule->getStateComplete();
	EMStatus->StateCurrent = static_cast<EMPackMLStateEnum>(pPackMLModule->getCurrentState());
	EMStatus->SubStateCurrent = pPackMLModule->getCurrentSubState();
	strcpy(EMStatus->StateInfo, pPackMLModule->getStateInfo());

	return true;
}

unsigned long EMGetParentAdr(unsigned long EmAddress){

	if(EmAddress == 0){
		return 0;
	}
	return reinterpret_cast<unsigned long int>(reinterpret_cast<PackMLModule*>(EmAddress)->getParentPtr());
		}
unsigned long EMGetChildrenAdrByIdx(unsigned long EmAddress, unsigned long EmIdx){

	if(EmAddress == 0){
		return 0;
	}

	return reinterpret_cast<unsigned long int>(reinterpret_cast<PackMLModule*>(EmAddress)->getChildPtr(EmIdx));

		}
unsigned long EMGetSiblingAdrByIdx(unsigned long EmAddress, unsigned long EmIdx){

	if(EmAddress == 0){
		return 0;
	}

	return reinterpret_cast<unsigned long int>(reinterpret_cast<PackMLModule*>(EmAddress)->getSiblingPtr(EmIdx));

		}
unsigned long EMGetRootAdrByIdx(unsigned long EmIdx){

	return reinterpret_cast<unsigned long int>(pPackMLModuleTable->getRootModuleByIdx(EmIdx));

}
unsigned long EMGetUserDataAdr(unsigned long EmAddress){

	if(EmAddress == 0){
		return 0;
	}
	return reinterpret_cast<unsigned long int>(reinterpret_cast<PackMLModule*>(EmAddress)->getUserMemoryPtr());

		}

plcbit EMSetCommand(unsigned long EmAddress, unsigned long EmAddressInterrupter, enum EMPackMLCmdEnum Command){

	if(EmAddress == 0){
		return false;
	}

	PackMLModule* pPackMLModule = reinterpret_cast<PackMLModule*>(EmAddress);

	switch(Command){

		case CMD_ABORT:
			pPackMLModule->setCmdAbort();
			break;

		case CMD_STOP:
			pPackMLModule->setCmdStop();
			break;

		case CMD_CLEAR:
			pPackMLModule->setCmdClear();
			break;

		case CMD_RESET:
			pPackMLModule->setCmdReset();
			break;

		case CMD_START:
			pPackMLModule->setCmdStart();
			break;

		case CMD_HOLD:
			pPackMLModule->setCmdHold();
			break;

		case CMD_UNHOLD:
			pPackMLModule->setCmdUnhold();
			break;

		case CMD_SUSPEND:
			pPackMLModule->setCmdSuspend();
			break;

		case CMD_UNSUSPEND:
			pPackMLModule->setCmdUnsuspend();
			break;

		case CMD_COMPLETE:
			pPackMLModule->setCmdComplete();
			break;

		case CMD_SC:
			pPackMLModule->setCmdStateComplete();
			break;

		default:
			return false;

	}

	if(EmAddressInterrupter == 0){
		pPackMLModule->setInteruptedBy(pPackMLModule);
	} else {
		pPackMLModule->setInteruptedBy(reinterpret_cast<PackMLModule*>(EmAddressInterrupter));
	}

	return true;

}

unsigned long EMGetModuleIdxByName(plcstring* EmName){

	if(EmName == nullptr){
		return 0xFFFFFFFF;
	}

	return pPackMLModuleTable->getModuleIndexByName(EmName);

}
```

#### EquipmentModule.cpp
```cpp
#include "BrdkPackML.h"
#include "../PackMLCore/PackMLModule.hpp"
#include "../PackMLCore/PackMLModuleTable.hpp"

extern unsigned long bur_heap_size;

extern PackMLModuleTable* pPackMLModuleTable;

// Main function. Is running cyclic together with FUB EquipmentModule()
void run(struct EquipmentModule* inst, PackMLModule* pPackMLModule)
{
	// Reading Setup structure
	pPackMLModule->setActivationCondition(static_cast<short int>(inst->Setup.ActivationCondition));
	pPackMLModule->setActivationPv(inst->Setup.Activate);

	pPackMLModule->setOverrideAbort(inst->Setup.Synchronisation.Override.Abort);
	pPackMLModule->setOverrideStop(inst->Setup.Synchronisation.Override.Stop);
	pPackMLModule->setOverrideComplete(inst->Setup.Synchronisation.Override.Complete);
	pPackMLModule->setOverrideSuspend(inst->Setup.Synchronisation.Override.Suspend);
	pPackMLModule->setOverrideUnsuspend(inst->Setup.Synchronisation.Override.Unsuspend);
	pPackMLModule->setOverrideHold(inst->Setup.Synchronisation.Override.Hold);
	pPackMLModule->setOverrideUnhold(inst->Setup.Synchronisation.Override.Unhold);
	pPackMLModule->setOverrideClear(inst->Setup.Synchronisation.Override.Clear);
	pPackMLModule->setOverrideReset(inst->Setup.Synchronisation.Override.Reset);
	pPackMLModule->setOverrideStart(inst->Setup.Synchronisation.Override.Start);

	pPackMLModule->setReactToAbort(inst->Setup.Synchronisation.ReactTo.Abort);
	pPackMLModule->setReactToStop(inst->Setup.Synchronisation.ReactTo.Stop);
	pPackMLModule->setReactToComplete(inst->Setup.Synchronisation.ReactTo.Complete);
	pPackMLModule->setReactToSuspend(inst->Setup.Synchronisation.ReactTo.Suspend);
	pPackMLModule->setReactToUnsuspend(inst->Setup.Synchronisation.ReactTo.Unsuspend);
	pPackMLModule->setReactToHold(inst->Setup.Synchronisation.ReactTo.Hold);
	pPackMLModule->setReactToUnhold(inst->Setup.Synchronisation.ReactTo.Unhold);
	pPackMLModule->setReactToClear(inst->Setup.Synchronisation.ReactTo.Clear);
	pPackMLModule->setReactToReset(inst->Setup.Synchronisation.ReactTo.Reset);
	pPackMLModule->setReactToStart(inst->Setup.Synchronisation.ReactTo.Start);

	pPackMLModule->setEscalateAbort(inst->Setup.Synchronisation.Escalate.Abort);
	pPackMLModule->setEscalateStop(inst->Setup.Synchronisation.Escalate.Stop);
	pPackMLModule->setEscalateComplete(inst->Setup.Synchronisation.Escalate.Complete);
	pPackMLModule->setEscalateSuspend(inst->Setup.Synchronisation.Escalate.Suspend);
	pPackMLModule->setEscalateUnsuspend(inst->Setup.Synchronisation.Escalate.Unsuspend);
	pPackMLModule->setEscalateHold(inst->Setup.Synchronisation.Escalate.Hold);
	pPackMLModule->setEscalateUnhold(inst->Setup.Synchronisation.Escalate.Unhold);
	pPackMLModule->setEscalateClear(inst->Setup.Synchronisation.Escalate.Clear);
	pPackMLModule->setEscalateReset(inst->Setup.Synchronisation.Escalate.Reset);
	pPackMLModule->setEscalateStart(inst->Setup.Synchronisation.Escalate.Start);

	if (inst->Info.OnStateEntry){
		inst->Info.OnStateEntry = false;
	}
	if (inst->Info.OnSubStateEntry){
		inst->Info.OnSubStateEntry = false;
	}

	long int oldSubstate = pPackMLModule->getCurrentSubState();
	if(oldSubstate != inst->SubState){
		if(inst->Setup.AuditSubStateChange){

			for(unsigned short int i = 0; i < EM_MAX_AUDIT_ENTRIES; i++){
				strcpy(inst->Info.Last[EM_MAX_AUDIT_ENTRIES - i], inst->Info.Last[(EM_MAX_AUDIT_ENTRIES - 1) - i]);
			}
			sprintf(inst->Info.Last[0], "Substate: %ld, time: %2.1f s.", oldSubstate, inst->Info.TimeInSubState);
		}
		pPackMLModule->setCurrentSubState(inst->SubState);
		inst->Info.OnSubStateEntry = true;
	}
	std::string oldStateInfo = pPackMLModule->getStateInfo();
	if(oldStateInfo != inst->StateInfo){
		pPackMLModule->setStateInfo(inst->StateInfo);
	}

	if(inst->SetModeID != inst->ModeID){
		// Restrict mode changes to certain states could be defined here: (-And also in the function EMSetMode())
		if (!pPackMLModule->setCurrentMode(inst->SetModeID)){
			inst->SetModeID = inst->ModeID;
		}

	}

	pPackMLModule->evaluateCmdAbort(inst->Command.Abort);
	pPackMLModule->evaluateCmdStop(inst->Command.Stop);
	pPackMLModule->evaluateCmdClear(inst->Command.Clear);
	pPackMLModule->evaluateCmdReset(inst->Command.Reset);
	pPackMLModule->evaluateCmdStart(inst->Command.Start);
	pPackMLModule->evaluateCmdSuspend(inst->Command.Suspend);
	pPackMLModule->evaluateCmdUnsuspend(inst->Command.Unsuspend);
	pPackMLModule->evaluateCmdHold(inst->Command.Hold);
	pPackMLModule->evaluateCmdUnhold(inst->Command.Unhold);
	pPackMLModule->evaluateCmdComplete(inst->Command.Complete);
	pPackMLModule->evaluateCmdStateComplete(inst->Command.StateComplete);

	if(inst->Setup.SkipStopStateComplete && pPackMLModule->getCmdStop()){
		pPackMLModule->setCmdStateComplete();
	}

	//--- End of things to handle before EM is being executed from lib on heap ---//

	// Run the packmlmodule service
	pPackMLModule->runPackMLModule();

	EMPackMLStateEnum stateCurrent = static_cast<EMPackMLStateEnum>(pPackMLModule->getCurrentState());
	// Update the FB info
	// State info
	if (inst->StateCurrent != stateCurrent) {

		if(inst->Setup.AuditStateChange){
			plcstring* oldStateStr = (plcstring*)pPackMLModule->getStateStr(static_cast<PackMLModuleStateEnu>(inst->StateCurrent));

			for(unsigned short int i = 0; i < EM_MAX_AUDIT_ENTRIES; i++){
				strcpy(inst->Info.Last[EM_MAX_AUDIT_ENTRIES - i], inst->Info.Last[(EM_MAX_AUDIT_ENTRIES - 1) - i]);
			}
			sprintf(inst->Info.Last[0], "State: %s, time: %2.1f s.", oldStateStr, inst->Info.TimeInState);
		}

		inst->StateCurrent = stateCurrent;

		inst->SubState = 0;
		pPackMLModule->setCurrentSubState(inst->SubState);
		inst->StateInfo[0] = 0;
		inst->Info.OnStateEntry = true;
		inst->Info.OnSubStateEntry = true;

		// Reset Cmds
		memset(&inst->Command, 0, sizeof(inst->Command));

	}

	inst->Info.TimeInState = pPackMLModule->getTimeInState();
	inst->Info.TimeInSubState = pPackMLModule->getTimeInSubState();

	inst->Info.ParentStateCurrent = static_cast<EMPackMLStateEnum>(pPackMLModule->getParentCurrentState());

	// Parent / Child / Sibling state/substate info
	inst->Info.ParentStateComplete = pPackMLModule->getParentStateComplete();
	inst->Info.SiblingsStateComplete = pPackMLModule->getSiblingsStateComplete();
	inst->Info.ChildrenStateComplete = pPackMLModule->getChildrenStateComplete();

	inst->Info.Level = pPackMLModule->getHierarchyLevel();
	inst->Info.ChildCount = pPackMLModule->getChildCount();
	inst->Info.SiblingCount = pPackMLModule->getSiblingCount();

	// Mode info
	if (inst->ModeID != pPackMLModule->getCurrentMode()) {

		if(inst->Setup.AuditStateChange){

			for(unsigned short int i = 0; i < EM_MAX_AUDIT_ENTRIES; i++){
				strcpy(inst->Info.Last[EM_MAX_AUDIT_ENTRIES - i], inst->Info.Last[(EM_MAX_AUDIT_ENTRIES - 1) - i]);
			}
			sprintf(inst->Info.Last[0], "ModeID: %d --> %ld", inst->ModeID, pPackMLModule->getCurrentMode());
		}

		inst->ModeID = static_cast<EMPackMLModeEnum>(pPackMLModule->getCurrentMode());
		inst->SetModeID = inst->ModeID ;

		inst->SubState = 0;
		pPackMLModule->setCurrentSubState(inst->SubState);
		inst->StateInfo[0] = 0;
	}

	if(inst->Setup.EnableInteruptedBy){
		PackMLModuleSharedInfo* pInteruptedBy =  pPackMLModule->getInteruptedByPtr();
		if(pInteruptedBy != nullptr){
			inst->Info.InteruptedBy.ModeID = inst->ModeID;
			inst->Info.InteruptedBy.StateCurrent = static_cast<EMPackMLStateEnum>(pInteruptedBy->getStateCurrent());
			inst->Info.InteruptedBy.SubStateCurrent = pInteruptedBy->getSubStateCurrent();
			inst->Info.InteruptedBy.StateComplete = pInteruptedBy->getStateComplete();
			strcpy(inst->Info.InteruptedBy.Name, pInteruptedBy->getName());
			strcpy(inst->Info.InteruptedBy.StateInfo, pInteruptedBy->getStateInfo());
		}
	}

	if(inst->Setup.EnableWaitingFor){
		PackMLModuleSharedInfo* pWaitingFor =  pPackMLModule->getWaitingForPtr();
		if(pWaitingFor != nullptr){
			inst->Info.WaitingFor.ModeID = inst->ModeID;
			inst->Info.WaitingFor.StateCurrent = static_cast<EMPackMLStateEnum>(pWaitingFor->getStateCurrent());
			inst->Info.WaitingFor.SubStateCurrent = pWaitingFor->getSubStateCurrent();
			inst->Info.WaitingFor.StateComplete = pWaitingFor->getStateComplete();
			strcpy(inst->Info.WaitingFor.Name, pWaitingFor->getName());
			strcpy(inst->Info.WaitingFor.StateInfo, pWaitingFor->getStateInfo());
		}
	}

	if(inst->Interface.Enable){
		inst->Internal.oldPubSubEnable = true;

		memcpy(reinterpret_cast<EMUserDataPubSubType*>(inst->Internal.userDataAddress), reinterpret_cast<EMUserDataPubSubType*>(&inst->Interface.Publish), sizeof(EMUserDataPubSubType));

		for(unsigned short int i = 0; i < EM_MAX_SUBSCRIPTIONS + 1; i++){

			if(inst->Interface.SubscriptionValid[i]){
				memcpy(reinterpret_cast<EMUserDataPubSubType*>(&inst->Interface.Subscribe[i]), reinterpret_cast<EMUserDataPubSubType*>(inst->Internal.subscriptionUserDataAddress[i]), sizeof(EMUserDataPubSubType));
			}

			if(strcmp(inst->Interface.SubscriptionEMName[i], inst->Internal.subscribedToEMName[i]) != 0){
				PackMLModule* pSubscribtionEm = pPackMLModuleTable->getModuleByName(inst->Interface.SubscriptionEMName[i]);
				if(pSubscribtionEm != nullptr){
					inst->Internal.subscriptionUserDataAddress[i] = reinterpret_cast<unsigned long int>(pSubscribtionEm->getUserMemoryPtr());
					inst->Interface.SubscriptionValid[i] = true;
					strcpy(inst->Internal.subscribedToEMName[i], inst->Interface.SubscriptionEMName[i]);
				} else {
					inst->Interface.SubscriptionValid[i] = false;
					inst->Internal.subscriptionUserDataAddress[i] = 0;
					inst->Internal.subscribedToEMName[i][0] = 0;
				}

				memset(reinterpret_cast<EMUserDataPubSubType*>(&inst->Interface.Subscribe[i]), 0, sizeof(EMUserDataPubSubType));

			}

		}
	} else if(not inst->Interface.Enable && inst->Internal.oldPubSubEnable){
		inst->Internal.oldPubSubEnable = false;
		memset(reinterpret_cast<EMUserDataPubSubType*>(&inst->Interface.Subscribe), 0, sizeof(EMUserDataPubSubType) * (EM_MAX_SUBSCRIPTIONS + 1));
		memset(reinterpret_cast<bool*>(&inst->Interface.SubscriptionValid), 0, sizeof(bool) * (EM_MAX_SUBSCRIPTIONS + 1));
		memset(reinterpret_cast<unsigned long int*>(&inst->Internal.subscriptionUserDataAddress), 0, sizeof(unsigned long int) * (EM_MAX_SUBSCRIPTIONS + 1));
		memset(reinterpret_cast<char*>(&inst->Internal.subscribedToEMName), 0, 256 * (EM_MAX_SUBSCRIPTIONS + 1));
	}

}

// ------------ IEC Functions and Function Blocks -----------------------------------------

void EquipmentModule(struct EquipmentModule* inst)
{

	// Initialize the module
	switch(inst->Internal.state){

		case 0:
			{
				// get name
				if(strlen(inst->Setup.Name) == 0){
					ST_name(0, inst->Setup.Name, 0);
				}

				char moduleName[256] = {""};

				if (inst->Setup.NameIndex == EM_MAX_NAME_INDEX){
					strcpy(moduleName, inst->Setup.Name);
				} else {
					sprintf(moduleName, "%s%d", inst->Setup.Name, inst->Setup.NameIndex);
				}

				// check if object exists
				PackMLModule* pPackMLModule = pPackMLModuleTable->getModuleByName(moduleName);

				// Create a new module if not exists
				if(pPackMLModule == nullptr){
					RTInfo_typ RTInfo_0;
					RTInfo_0.enable = 1;
					RTInfo(&RTInfo_0);

					pPackMLModule = new PackMLModule(moduleName);
					pPackMLModule->setCycleTime(static_cast<float>(RTInfo_0.cycle_time) * 0.000001);
					inst->Info.CycleTime = static_cast<float>(RTInfo_0.cycle_time) * 0.000001;

					// Create userData for misc usage e.g. sync and priority, and get pointer.
					inst->Internal.userDataAddress = reinterpret_cast<unsigned long int>(pPackMLModule->createUserMemory(sizeof(EMUserDataPubSubType)));
					inst->Internal.state = 20;
				} else {
					// We should copy all the options from the heap to the IEC on stack
					strcpy(inst->Setup.ParentName, pPackMLModule->getParentName());
					strcpy(inst->Info.ParentName, inst->Setup.ParentName);

					inst->Internal.userDataAddress = reinterpret_cast<unsigned long int>(pPackMLModule->getUserMemoryPtr());
					inst->Info.EmIndex = pPackMLModuleTable->getModuleIndexByName(moduleName);

					inst->Internal.state = 40;
				}

				inst->Internal.emAddress = reinterpret_cast<unsigned long int>(pPackMLModule);
				inst->Info.EmAddress = inst->Internal.emAddress;
				inst->Info.UserDataAddress = inst->Internal.userDataAddress;
				strcpy(inst->Info.EmName, moduleName);

			}
			break;

		case 20: // register the object
			if(pPackMLModuleTable->registerEm(inst->Internal.emAddress, &inst->Info.EmIndex)){
				inst->Internal.state = 30;
			}
			break;

		case 30: // Init EM phase // interlinking
			{
				PackMLModule* pPackMLModule = reinterpret_cast<PackMLModule*>(inst->Internal.emAddress);

				if(strlen(inst->Setup.ParentName) > 0){
					inst->Internal.state = 35;
				} else {
					pPackMLModule->initModule();
					inst->Internal.state = 40;
				}
				strcpy(inst->Info.ParentName, inst->Setup.ParentName);

				// **** do we need it here?? test
				//				pPackMLModule->runPackMLModule();
			}
			break;

		case 35:
			{
				PackMLModule* pPackMLModule = reinterpret_cast<PackMLModule*>(inst->Internal.emAddress);
				// Can get stucked here --> **inst->Info.ParentName**
				if(strcmp(inst->Setup.ParentName, inst->Info.ParentName) != 0){
					inst->Internal.state = 30;
				} else if(pPackMLModule->initModule(reinterpret_cast<PackMLModule*>(pPackMLModuleTable->getModuleByName(inst->Info.ParentName)))){
					//					strcpy(inst->Info.ParentName, pPackMLModule->getParentName());
					inst->Internal.state = 40;
				}

			}
			break;

		case 40: // run state
			// if EmLinkParent changes reinitilise the module in state 30
			{
				PackMLModule* pPackMLModule = reinterpret_cast<PackMLModule*>(inst->Internal.emAddress);

				if(strcmp(inst->Setup.ParentName, inst->Info.ParentName) != 0){
					inst->Internal.state = 50;
				} else {
					run(inst, pPackMLModule);
				}

			}
			break;

		case 50: // exit module and go to state 10
			{
				PackMLModule* pPackMLModule = reinterpret_cast<PackMLModule*>(inst->Internal.emAddress);

				if(pPackMLModule->exitModule()){
					inst->Internal.state = 30;

					if(inst->Setup.AuditStateChange){
						plcstring* oldStateStr = (plcstring*)pPackMLModule->getStateStr(static_cast<PackMLModuleStateEnu>(inst->StateCurrent));

						for(unsigned short int i = 0; i < EM_MAX_AUDIT_ENTRIES; i++){
							strcpy(inst->Info.Last[EM_MAX_AUDIT_ENTRIES - i], inst->Info.Last[(EM_MAX_AUDIT_ENTRIES - 1) - i]);
						}
						sprintf(inst->Info.Last[0], "State: %s, time: %2.1f s.", oldStateStr, inst->Info.TimeInState);
					}

					inst->Info.TimeInState = 0;
					inst->Info.ParentName[0] = 0;
					inst->Info.ParentStateCurrent = STATE_UNDEFINED;
					inst->Info.ParentStateComplete = false;
					inst->Info.Level = 0;
					inst->Info.SiblingCount = 1;
					inst->StateCurrent = STATE_UNDEFINED;
					inst->SubState = 0;
					inst->StateInfo[0] = 0;
					memset(&inst->Command, 0, sizeof(inst->Command));
				}

			}
			break;
	}

}
```

#### ControlModule.cpp
```cpp
#include "BrdkPackML.h"
#include "../PackMLCore/PackMLModule.hpp"
#include "../PackMLCore/PackMLModuleTable.hpp"

extern unsigned long bur_heap_size;

extern PackMLModuleTable* pPackMLModuleTable;

// Main function. Is running cyclic together with FUB EquipmentModule()
void run(struct ControlModule* inst, PackMLModule* pPackMLModule)
{

	if (inst->Info.OnStateEntry){
		inst->Info.OnStateEntry = false;
	}
	if (inst->Info.OnSubStateEntry){
		inst->Info.OnSubStateEntry = false;
	}

	if(inst->Internal.oldSubState != inst->SubState){
		if(inst->Setup.AuditSubStateChange){

			for(unsigned short int i = 0; i < EM_MAX_AUDIT_ENTRIES; i++){
				strcpy(inst->Info.Last[EM_MAX_AUDIT_ENTRIES - i], inst->Info.Last[(EM_MAX_AUDIT_ENTRIES - 1) - i]);
			}
			sprintf(inst->Info.Last[0], "Substate: %ld, time: %2.1f s.", inst->Internal.oldSubState, inst->Info.TimeInSubState);
		}
		inst->Internal.oldSubState = inst->SubState;
		inst->Info.TimeInSubState = 0.0;
		inst->Info.OnSubStateEntry = true;
	}

	// Update the FB info
	// State info
	if (inst->State != inst->Internal.oldState) {

		if(inst->Setup.AuditStateChange){

			for(unsigned short int i = 0; i < EM_MAX_AUDIT_ENTRIES; i++){
				strcpy(inst->Info.Last[EM_MAX_AUDIT_ENTRIES - i], inst->Info.Last[(EM_MAX_AUDIT_ENTRIES - 1) - i]);
			}
			sprintf(inst->Info.Last[0], "State: %ld, time: %2.1f s.", inst->Internal.oldState, inst->Info.TimeInState);
		}

		inst->Internal.oldState = inst->State;

		inst->SubState = 0;
		inst->Internal.oldSubState = 0;
		inst->StateInfo[0] = 0;
		inst->Info.TimeInState = 0.0;
		inst->Info.TimeInSubState = 0.0;
		inst->Info.OnStateEntry = true;
		inst->Info.OnSubStateEntry = true;

	}

	inst->Info.TimeInState += inst->Internal.cycleTime;
	inst->Info.TimeInSubState += inst->Internal.cycleTime;

	// Parent / Child / Sibling state/substate info
	if (pPackMLModule != nullptr){
		inst->Info.Level = pPackMLModule->getHierarchyLevel() + 1;
		inst->Info.ParentStateCurrent = static_cast<EMPackMLStateEnum>(pPackMLModule->getCurrentState());
	} else {
		inst->Info.Level = 0;
		inst->Info.ParentStateCurrent = STATE_UNDEFINED;
	}

	if(inst->Interface.Enable){
		inst->Internal.oldPubSubEnable = true;

		for(unsigned short int i = 0; i < EM_MAX_SUBSCRIPTIONS + 1; i++){

			if(inst->Interface.SubscriptionValid[i]){
				memcpy(reinterpret_cast<EMUserDataPubSubType*>(&inst->Interface.Subscribe[i]), reinterpret_cast<EMUserDataPubSubType*>(inst->Internal.subscriptionUserDataAddress[i]), sizeof(EMUserDataPubSubType));
			}

			if(strcmp(inst->Interface.SubscriptionEMName[i], inst->Internal.subscribedToEMName[i]) != 0){
				PackMLModule* pSubscribtionEm = pPackMLModuleTable->getModuleByName(inst->Interface.SubscriptionEMName[i]);
				if(pSubscribtionEm != nullptr){
					inst->Internal.subscriptionUserDataAddress[i] = reinterpret_cast<unsigned long int>(pSubscribtionEm->getUserMemoryPtr());
					inst->Interface.SubscriptionValid[i] = true;
					strcpy(inst->Internal.subscribedToEMName[i], inst->Interface.SubscriptionEMName[i]);
				} else {
					inst->Interface.SubscriptionValid[i] = false;
					inst->Internal.subscriptionUserDataAddress[i] = 0;
					inst->Internal.subscribedToEMName[i][0] = 0;
				}

				memset(reinterpret_cast<EMUserDataPubSubType*>(&inst->Interface.Subscribe[i]), 0, sizeof(EMUserDataPubSubType));

			}

		}
	} else if(not inst->Interface.Enable && inst->Internal.oldPubSubEnable){
		inst->Internal.oldPubSubEnable = false;
		memset(reinterpret_cast<EMUserDataPubSubType*>(&inst->Interface.Subscribe), 0, sizeof(EMUserDataPubSubType) * (EM_MAX_SUBSCRIPTIONS + 1));
		memset(reinterpret_cast<bool*>(&inst->Interface.SubscriptionValid), 0, sizeof(bool) * (EM_MAX_SUBSCRIPTIONS + 1));
		memset(reinterpret_cast<unsigned long int*>(&inst->Internal.subscriptionUserDataAddress), 0, sizeof(unsigned long int) * (EM_MAX_SUBSCRIPTIONS + 1));
		memset(reinterpret_cast<char*>(&inst->Internal.subscribedToEMName), 0, 256 * (EM_MAX_SUBSCRIPTIONS + 1));
	}

}

// ------------ IEC Functions and Function Blocks -----------------------------------------

void ControlModule(struct ControlModule* inst)
{

	// Initialize the module
	switch(inst->Internal.state){

		case 0:
			{
				// get name
				if(strlen(inst->Setup.Name) == 0){
					ST_name(0, inst->Setup.Name, 0);
				}

				char moduleName[256] = {""};

				if (inst->Setup.NameIndex == EM_MAX_NAME_INDEX){
					strcpy(moduleName, inst->Setup.Name);
				} else {
					sprintf(moduleName, "%s%d", inst->Setup.Name, inst->Setup.NameIndex);
				}

				strcpy(inst->Info.CmName, moduleName);

				RTInfo_typ RTInfo_0;
				RTInfo_0.enable = 1;
				RTInfo(&RTInfo_0);
				inst->Internal.cycleTime = static_cast<float>(RTInfo_0.cycle_time) * 0.000001;
				inst->Info.CycleTime = inst->Internal.cycleTime;
				inst->Internal.state = 30;
			}
			break;

		case 30: // Init EM phase // interlinking
			{
				if(strlen(inst->Setup.ParentName) > 0){
					inst->Internal.state = 35;
				} else {
					inst->Internal.state = 40;
				}
				strcpy(inst->Info.ParentName, inst->Setup.ParentName);
			}
			break;

		case 35:
			{

				PackMLModule* pPackMLModule = pPackMLModuleTable->getModuleByName(inst->Info.ParentName);

				if(strcmp(inst->Setup.ParentName, inst->Info.ParentName) != 0){
					inst->Internal.state = 30;

				} else if(pPackMLModule != nullptr){
					inst->Internal.parentEmAddress = reinterpret_cast<unsigned long int>(pPackMLModule);
					inst->Info.ParentEmAddress = inst->Internal.parentEmAddress;
					inst->Info.ParentEmIndex = pPackMLModuleTable->getModuleIndexByName(inst->Info.ParentName);
					inst->Internal.state = 40;
				}

			}
			break;

		case 40: // run state
			// if EmLinkParent changes reinitilise the module in state 30
			{
				PackMLModule* pPackMLModule = reinterpret_cast<PackMLModule*>(inst->Internal.parentEmAddress);

				if(strcmp(inst->Setup.ParentName, inst->Info.ParentName) != 0){
					inst->Info.ParentName[0] = 0;
					inst->Info.ParentEmAddress = 0;
					inst->Info.ParentEmIndex = 0;
					inst->Internal.parentEmAddress = 0;
					inst->Internal.state = 30;
				}
				run(inst, pPackMLModule);
			}
			break;
	}

}
```

### Library Logical/Libraries/brdkSTR (ANSIC, version 1.8.0)
Depends on: astime
